C01807=1145.938,166.654,-59.645,-178.486,7.082,148.879
C01808=1145.942,166.405,-59.623,-178.489,7.080,148.879
C01809=1145.947,166.156,-59.601,-178.492,7.077,148.880
C01810=1145.951,165.907,-59.579,-178.495,7.076,148.880
C01811=1145.956,165.658,-59.558,-178.497,7.074,148.880
C01812=1145.961,165.409,-59.535,-178.500,7.071,148.881
C01813=1145.966,165.160,-59.513,-178.503,7.069,148.881
C01814=1145.970,164.911,-59.491,-178.506,7.068,148.881
C01815=1145.975,164.662,-59.469,-178.509,7.065,148.882
C01816=1145.980,164.413,-59.447,-178.511,7.063,148.882
C01817=1145.984,164.165,-59.425,-178.514,7.061,148.882
C01818=1145.988,163.915,-59.403,-178.517,7.059,148.883
C01819=1145.993,163.667,-59.381,-178.520,7.057,148.883
C01820=1145.998,163.417,-59.359,-178.522,7.055,148.883
C01821=1146.003,163.168,-59.337,-178.525,7.052,148.883
C01822=1146.008,162.919,-59.316,-178.528,7.051,148.884
C01823=1146.013,162.670,-59.294,-178.531,7.049,148.884
C01824=1146.017,162.421,-59.272,-178.534,7.046,148.885
C01825=1146.022,162.172,-59.250,-178.536,7.044,148.885
C01826=1146.027,161.923,-59.229,-178.539,7.043,148.885
C01827=1146.031,161.674,-59.206,-178.542,7.040,148.885
C01828=1146.036,161.425,-59.185,-178.545,7.038,148.886
C01829=1146.040,161.176,-59.163,-178.548,7.037,148.886
C01830=1146.045,160.927,-59.141,-178.550,7.034,148.886
C01831=1146.050,160.679,-59.119,-178.553,7.032,148.887
C01832=1146.054,160.429,-59.097,-178.556,7.030,148.887
C01833=1146.059,160.180,-59.076,-178.559,7.029,148.887
C01834=1146.064,159.931,-59.054,-178.562,7.026,148.888
C01835=1146.068,159.682,-59.033,-178.564,7.024,148.888
C01836=1146.073,159.433,-59.011,-178.567,7.022,148.888
C01837=1146.078,159.184,-58.989,-178.570,7.020,148.889
C01838=1146.083,158.935,-58.968,-178.573,7.018,148.889
C01839=1146.088,158.686,-58.946,-178.575,7.016,148.889
C01840=1146.092,158.437,-58.924,-178.578,7.013,148.890
C01841=1146.097,158.188,-58.903,-178.581,7.012,148.890
C01842=1146.101,157.919,-58.880,-178.584,7.010,148.890
C01843=1146.107,157.650,-58.856,-178.587,7.007,148.891
C01844=1146.111,157.381,-58.833,-178.590,7.006,148.891
C01845=1146.117,157.112,-58.810,-178.593,7.003,148.891
C01846=1146.122,156.863,-58.788,-178.596,7.001,148.892
C01847=1146.126,156.613,-58.767,-178.599,6.999,148.892
C01848=1146.130,156.365,-58.745,-178.602,6.997,148.893
C01849=1146.135,156.116,-58.724,-178.604,6.995,148.893
C01850=1146.140,155.867,-58.703,-178.607,6.993,148.893
C01851=1146.145,155.618,-58.681,-178.610,6.991,148.893
C01852=1146.150,155.369,-58.660,-178.613,6.989,148.894
C01853=1146.155,155.120,-58.638,-178.615,6.987,148.894
C01854=1146.159,154.871,-58.616,-178.618,6.986,148.895
C01855=1146.163,154.622,-58.596,-178.621,6.983,148.895
C01856=1146.168,154.373,-58.574,-178.624,6.981,148.895
C01857=1146.174,154.124,-58.553,-178.626,6.979,148.895
C01858=1146.178,153.874,-58.531,-178.629,6.978,148.896
C01859=1146.183,153.625,-58.510,-178.632,6.975,148.896
C01860=1146.187,153.377,-58.489,-178.635,6.973,148.897
C01861=1146.192,153.128,-58.468,-178.638,6.972,148.897
C01862=1146.197,152.878,-58.446,-178.640,6.970,148.897
C01863=1146.202,152.629,-58.425,-178.643,6.967,148.898
C01864=1146.207,152.380,-58.403,-178.646,6.965,148.898
C01865=1146.211,152.131,-58.383,-178.649,6.964,148.898
C01866=1146.215,151.882,-58.361,-178.651,6.962,148.899
C01867=1146.220,151.633,-58.340,-178.655,6.959,148.899
C01868=1146.225,151.384,-58.319,-178.657,6.958,148.899
C01869=1146.230,151.135,-58.298,-178.660,6.956,148.900
C01870=1146.235,150.886,-58.277,-178.662,6.954,148.900
C01871=1146.239,150.637,-58.255,-178.666,6.951,148.900
C01872=1146.244,150.388,-58.234,-178.668,6.950,148.901
C01873=1146.249,150.138,-58.213,-178.671,6.948,148.901
C01874=1146.254,149.890,-58.192,-178.674,6.946,148.901
C01875=1146.258,149.641,-58.171,-178.676,6.945,148.902
C01876=1146.263,149.392,-58.150,-178.680,6.942,148.902
C01877=1146.268,149.142,-58.128,-178.682,6.940,148.902
C01878=1146.272,148.893,-58.108,-178.685,6.938,148.903
C01879=1146.277,148.644,-58.087,-178.687,6.936,148.903
C01880=1146.282,148.395,-58.065,-178.690,6.935,148.904
C01881=1146.286,148.146,-58.045,-178.693,6.932,148.904
C01882=1146.292,147.897,-58.024,-178.696,6.931,148.904
C01883=1146.296,147.648,-58.004,-178.699,6.929,148.905
C01884=1146.300,147.399,-57.982,-178.701,6.927,148.905
C01885=1146.306,147.150,-57.961,-178.705,6.925,148.905
C01886=1146.310,146.901,-57.940,-178.707,6.923,148.906
C01887=1146.315,146.651,-57.919,-178.710,6.921,148.906
C01888=1146.319,146.403,-57.898,-178.712,6.919,148.906
C01889=1146.324,146.154,-57.877,-178.715,6.917,148.907
C01890=1146.329,145.905,-57.857,-178.718,6.916,148.907
C01891=1146.334,145.656,-57.836,-178.721,6.913,148.907
C01892=1146.339,145.407,-57.816,-178.724,6.911,148.908
C01893=1146.344,145.157,-57.795,-178.727,6.910,148.908
C01894=1146.348,144.907,-57.773,-178.729,6.908,148.909
C01895=1146.352,144.659,-57.752,-178.732,6.906,148.909
C01896=1146.358,144.410,-57.731,-178.735,6.904,148.909
C01897=1146.362,144.161,-57.711,-178.738,6.902,148.910
C01898=1146.366,143.912,-57.690,-178.740,6.900,148.910
C01899=1146.372,143.663,-57.670,-178.743,6.898,148.910
C01900=1146.376,143.414,-57.649,-178.746,6.897,148.911
C01901=1146.381,143.164,-57.628,-178.748,6.895,148.911
C01902=1146.386,142.916,-57.608,-178.752,6.892,148.912
C01903=1146.391,142.666,-57.587,-178.754,6.891,148.912
C01904=1146.395,142.417,-57.566,-178.757,6.889,148.912
C01905=1146.400,142.168,-57.545,-178.760,6.887,148.913
C01906=1146.405,141.919,-57.525,-178.763,6.885,148.913
C01907=1146.409,141.670,-57.505,-178.765,6.884,148.913
C01908=1146.415,141.421,-57.484,-178.769,6.881,148.914
C01909=1146.419,141.172,-57.463,-178.771,6.879,148.914
C01910=1146.424,140.923,-57.442,-178.774,6.878,148.915
C01911=1146.429,140.674,-57.422,-178.777,6.876,148.915
C01912=1146.433,140.425,-57.402,-178.779,6.874,148.915
C01913=1146.438,140.176,-57.381,-178.782,6.873,148.916
C01914=1146.443,139.926,-57.361,-178.784,6.871,148.916
C01915=1146.447,139.677,-57.341,-178.788,6.868,148.916
C01916=1146.453,139.428,-57.320,-178.790,6.866,148.917
C01917=1146.457,139.179,-57.299,-178.793,6.865,148.917
C01918=1146.461,138.930,-57.279,-178.796,6.863,148.917
C01919=1146.467,138.681,-57.258,-178.799,6.861,148.918
C01920=1146.471,138.432,-57.238,-178.801,6.859,148.918
C01921=1146.476,138.182,-57.218,-178.804,6.858,148.919
C01922=1146.481,137.933,-57.197,-178.807,6.855,148.919
C01923=1146.485,137.684,-57.177,-178.810,6.854,148.919
C01924=1146.490,137.435,-57.156,-178.813,6.852,148.920
C01925=1146.494,137.186,-57.136,-178.815,6.850,148.920
C01926=1146.500,136.936,-57.116,-178.818,6.848,148.921
C01927=1146.505,136.688,-57.096,-178.821,6.847,148.921
C01928=1146.509,136.439,-57.075,-178.824,6.845,148.921
C01929=1146.515,136.189,-57.055,-178.826,6.843,148.922
C01930=1146.519,135.940,-57.035,-178.830,6.841,148.922
C01931=1146.524,135.691,-57.014,-178.832,6.839,148.923
C01932=1146.528,135.442,-56.994,-178.835,6.837,148.923
C01933=1146.533,135.193,-56.974,-178.838,6.836,148.923
C01934=1146.538,134.943,-56.953,-178.840,6.834,148.924
C01935=1146.542,134.694,-56.933,-178.843,6.832,148.924
C01936=1146.548,134.446,-56.914,-178.846,6.831,148.925
C01937=1146.552,134.197,-56.893,-178.849,6.829,148.925
C01938=1146.557,133.947,-56.874,-178.851,6.827,148.925
C01939=1146.562,133.698,-56.853,-178.854,6.825,148.926
C01940=1146.566,133.449,-56.832,-178.857,6.823,148.926
C01941=1146.571,133.199,-56.813,-178.860,6.821,148.926
C01942=1146.576,132.950,-56.792,-178.863,6.819,148.927
C01943=1146.581,132.701,-56.773,-178.865,6.818,148.927
C01944=1146.585,132.452,-56.753,-178.868,6.816,148.928
C01945=1146.590,132.203,-56.733,-178.871,6.814,148.928
C01946=1146.596,131.935,-56.711,-178.874,6.813,148.928
C01947=1146.600,131.666,-56.689,-178.877,6.810,148.929
C01948=1146.606,131.397,-56.668,-178.880,6.808,148.929
C01949=1146.611,131.129,-56.646,-178.882,6.807,148.930
C01950=1146.615,130.879,-56.626,-178.885,6.805,148.930
C01951=1146.620,130.630,-56.606,-178.888,6.803,148.930
C01952=1146.625,130.382,-56.587,-178.890,6.802,148.931
C01953=1146.630,130.133,-56.566,-178.894,6.799,148.931
C01954=1146.635,129.883,-56.546,-178.897,6.797,148.932
C01955=1146.640,129.633,-56.526,-178.900,6.796,148.932
C01956=1146.645,129.385,-56.506,-178.902,6.794,148.933
C01957=1146.650,129.135,-56.487,-178.905,6.793,148.933
C01958=1146.654,128.886,-56.466,-178.908,6.791,148.933
C01959=1146.659,128.637,-56.447,-178.911,6.789,148.934
C01960=1146.664,128.388,-56.427,-178.913,6.788,148.934
C01961=1146.669,128.139,-56.407,-178.916,6.786,148.935
C01962=1146.673,127.889,-56.387,-178.919,6.784,148.935
C01963=1146.678,127.640,-56.368,-178.921,6.782,148.935
C01964=1146.683,127.392,-56.348,-178.924,6.781,148.936
C01965=1146.688,127.142,-56.328,-178.927,6.779,148.936
C01966=1146.693,126.892,-56.308,-178.930,6.777,148.937
C01967=1146.696,126.644,-56.289,-178.932,6.776,148.937
C01968=1146.702,126.395,-56.269,-178.935,6.774,148.937
C01969=1146.706,126.145,-56.250,-178.938,6.772,148.938
C01970=1146.711,125.896,-56.230,-178.940,6.771,148.938
C01971=1146.716,125.648,-56.210,-178.943,6.769,148.939
C01972=1146.721,125.398,-56.190,-178.947,6.766,148.939
C01973=1146.726,125.148,-56.171,-178.949,6.765,148.939
C01974=1146.731,124.900,-56.151,-178.952,6.763,148.940
C01975=1146.735,124.651,-56.131,-178.955,6.761,148.940
C01976=1146.740,124.401,-56.111,-178.957,6.760,148.941
C01977=1146.746,124.152,-56.092,-178.960,6.758,148.941
C01978=1146.750,123.903,-56.073,-178.963,6.756,148.941
C01979=1146.754,123.653,-56.053,-178.966,6.754,148.942
C01980=1146.760,123.404,-56.034,-178.969,6.753,148.942
C01981=1146.764,123.156,-56.014,-178.971,6.751,148.943
C01982=1146.769,122.906,-55.994,-178.974,6.750,148.943
C01983=1146.774,122.657,-55.975,-178.977,6.748,148.944
C01984=1146.778,122.408,-55.956,-178.980,6.746,148.944
C01985=1146.783,122.158,-55.936,-178.982,6.745,148.944
C01986=1146.788,121.909,-55.917,-178.985,6.743,148.945
C01987=1146.793,121.660,-55.897,-178.988,6.741,148.945
C01988=1146.798,121.411,-55.878,-178.991,6.739,148.946
C01989=1146.802,121.162,-55.859,-178.993,6.738,148.946
C01990=1146.807,120.912,-55.839,-178.996,6.736,148.946
C01991=1146.812,120.663,-55.820,-178.999,6.734,148.947
C01992=1146.817,120.414,-55.800,-179.001,6.733,148.947
C01993=1146.822,120.165,-55.781,-179.004,6.731,148.948
C01994=1146.827,119.916,-55.762,-179.007,6.730,148.948
C01995=1146.831,119.666,-55.742,-179.010,6.728,148.949
C01996=1146.837,119.417,-55.723,-179.013,6.726,148.949
C01997=1146.841,119.168,-55.704,-179.016,6.725,148.949
C01998=1146.846,118.919,-55.684,-179.018,6.723,148.950
C01999=1146.851,118.669,-55.665,-179.021,6.721,148.950
C02000=1146.856,118.421,-55.646,-179.024,6.719,148.951
C02001=1146.860,118.171,-55.626,-179.026,6.718,148.951
C02002=1146.865,117.922,-55.607,-179.029,6.716,148.951
C02003=1146.870,117.673,-55.588,-179.032,6.714,148.952
C02004=1146.874,117.423,-55.569,-179.035,6.713,148.952
C02005=1146.880,117.174,-55.550,-179.038,6.711,148.953
C02006=1146.885,116.925,-55.530,-179.040,6.710,148.953
C02007=1146.889,116.676,-55.512,-179.043,6.709,148.954
C02008=1146.894,116.426,-55.492,-179.045,6.707,148.954
C02009=1146.899,116.178,-55.473,-179.048,6.705,148.954
C02010=1146.903,115.928,-55.454,-179.051,6.704,148.955
C02011=1146.909,115.679,-55.435,-179.054,6.702,148.955
C02012=1146.913,115.430,-55.416,-179.056,6.700,148.956
C02013=1146.918,115.181,-55.397,-179.059,6.699,148.956
C02014=1146.923,114.931,-55.377,-179.062,6.697,148.956
C02015=1146.928,114.682,-55.359,-179.065,6.696,148.957
C02016=1146.933,114.432,-55.339,-179.068,6.694,148.958
C02017=1146.937,114.184,-55.321,-179.070,6.692,148.958
C02018=1146.943,113.935,-55.301,-179.073,6.690,148.958
C02019=1146.948,113.685,-55.282,-179.076,6.689,148.959
C02020=1146.952,113.436,-55.264,-179.079,6.687,148.959
C02021=1146.957,113.187,-55.244,-179.081,6.685,148.960
C02022=1146.962,112.937,-55.226,-179.084,6.684,148.960
C02023=1146.967,112.688,-55.206,-179.087,6.682,148.960
C02024=1146.971,112.439,-55.188,-179.090,6.681,148.961
C02025=1146.976,112.189,-55.169,-179.093,6.679,148.961
C02026=1146.981,111.941,-55.150,-179.095,6.678,148.962
C02027=1146.986,111.692,-55.131,-179.098,6.676,148.962
C02028=1146.991,111.442,-55.112,-179.100,6.675,148.963
C02029=1146.996,111.193,-55.093,-179.103,6.673,148.963
C02030=1147.000,110.943,-55.075,-179.106,6.671,148.963
C02031=1147.006,110.694,-55.055,-179.109,6.670,148.964
C02032=1147.010,110.446,-55.037,-179.112,6.668,148.964
C02033=1147.015,110.196,-55.018,-179.114,6.667,148.965
C02034=1147.020,109.947,-54.999,-179.117,6.665,148.965
C02035=1147.025,109.697,-54.980,-179.120,6.663,148.966
C02036=1147.029,109.448,-54.962,-179.123,6.662,148.966
C02037=1147.034,109.199,-54.944,-179.125,6.660,148.967
C02038=1147.039,108.949,-54.924,-179.128,6.659,148.967
C02039=1147.044,108.700,-54.906,-179.131,6.658,148.968
C02040=1147.049,108.451,-54.887,-179.133,6.656,148.968
C02041=1147.054,108.202,-54.868,-179.136,6.654,148.968
C02042=1147.058,107.953,-54.850,-179.139,6.653,148.969
C02043=1147.063,107.703,-54.831,-179.142,6.651,148.969
C02044=1147.068,107.454,-54.812,-179.144,6.649,148.970
C02045=1147.074,107.205,-54.793,-179.147,6.648,148.970
C02046=1147.078,106.955,-54.775,-179.150,6.646,148.971
C02047=1147.083,106.706,-54.756,-179.153,6.644,148.971
C02048=1147.088,106.457,-54.738,-179.155,6.644,148.971
C02049=1147.092,106.208,-54.719,-179.158,6.642,148.972
C02050=1147.097,105.939,-54.699,-179.161,6.641,148.973
C02051=1147.103,105.671,-54.679,-179.164,6.638,148.973
C02052=1147.108,105.403,-54.660,-179.167,6.636,148.973
C02053=1147.114,105.135,-54.639,-179.170,6.635,148.974
C02054=1147.118,104.885,-54.621,-179.173,6.633,148.974
C02055=1147.123,104.636,-54.603,-179.176,6.632,148.975
C02056=1147.128,104.387,-54.584,-179.178,6.631,148.975
C02057=1147.133,104.137,-54.566,-179.181,6.629,148.976
C02058=1147.137,103.888,-54.547,-179.183,6.627,148.976
C02059=1147.142,103.639,-54.529,-179.186,6.626,148.977
C02060=1147.148,103.390,-54.510,-179.189,6.624,148.977
C02061=1147.152,103.140,-54.492,-179.192,6.623,148.978
C02062=1147.157,102.891,-54.474,-179.195,6.621,148.978
C02063=1147.162,102.642,-54.455,-179.197,6.620,148.978
C02064=1147.167,102.392,-54.436,-179.200,6.619,148.979
C02065=1147.172,102.143,-54.418,-179.203,6.617,148.979
C02066=1147.176,101.893,-54.400,-179.205,6.616,148.980
C02067=1147.181,101.644,-54.382,-179.208,6.614,148.980
C02068=1147.187,101.395,-54.363,-179.211,6.612,148.981
C02069=1147.192,101.146,-54.345,-179.214,6.610,148.981
C02070=1147.196,100.896,-54.326,-179.216,6.610,148.981
C02071=1147.201,100.647,-54.308,-179.219,6.608,148.982
C02072=1147.206,100.398,-54.290,-179.222,6.607,148.983
C02073=1147.211,100.149,-54.272,-179.224,6.605,148.983
C02074=1147.216,99.899,-54.254,-179.227,6.603,148.983
C02075=1147.220,99.650,-54.235,-179.230,6.602,148.984
C02076=1147.225,99.401,-54.217,-179.233,6.600,148.984
C02077=1147.230,99.152,-54.199,-179.235,6.599,148.985
C02078=1147.235,98.903,-54.181,-179.238,6.598,148.985
C02079=1147.240,98.653,-54.163,-179.241,6.596,148.986
C02080=1147.244,98.403,-54.145,-179.244,6.594,148.986
C02081=1147.249,98.154,-54.127,-179.247,6.593,148.987
C02082=1147.254,97.905,-54.109,-179.249,6.592,148.987
C02083=1147.260,97.656,-54.090,-179.252,6.590,148.988
C02084=1147.265,97.406,-54.072,-179.254,6.589,148.988
C02085=1147.270,97.157,-54.054,-179.257,6.587,148.988
C02086=1147.274,96.908,-54.036,-179.260,6.586,148.989
C02087=1147.279,96.658,-54.018,-179.263,6.584,148.989
C02088=1147.284,96.409,-54.000,-179.265,6.583,148.990
C02089=1147.289,96.160,-53.982,-179.268,6.581,148.990
C02090=1147.294,95.911,-53.964,-179.271,6.580,148.991
C02091=1147.298,95.662,-53.946,-179.274,6.578,148.991
C02092=1147.303,95.412,-53.928,-179.277,6.577,148.992
C02093=1147.308,95.163,-53.910,-179.279,6.576,148.992
C02094=1147.313,94.914,-53.892,-179.281,6.574,148.993
C02095=1147.317,94.664,-53.874,-179.285,6.573,148.993
C02096=1147.323,94.414,-53.856,-179.287,6.571,148.994
C02097=1147.328,94.165,-53.838,-179.290,6.570,148.994
C02098=1147.333,93.916,-53.820,-179.292,6.569,148.994
C02099=1147.337,93.667,-53.802,-179.295,6.567,148.995
C02100=1147.342,93.418,-53.784,-179.298,6.566,148.996
C02101=1147.347,93.168,-53.766,-179.301,6.564,148.996
C02102=1147.352,92.919,-53.749,-179.304,6.562,148.996
C02103=1147.357,92.669,-53.731,-179.306,6.561,148.997
C02104=1147.362,92.420,-53.713,-179.309,6.560,148.997
C02105=1147.367,92.171,-53.695,-179.312,6.558,148.998
C02106=1147.372,91.922,-53.677,-179.314,6.557,148.998
C02107=1147.377,91.672,-53.660,-179.317,6.555,148.999
C02108=1147.382,91.423,-53.643,-179.319,6.554,148.999
C02109=1147.386,91.174,-53.625,-179.323,6.553,149.000
C02110=1147.391,90.925,-53.607,-179.325,6.551,149.000
C02111=1147.397,90.675,-53.589,-179.328,6.550,149.001
C02112=1147.401,90.426,-53.571,-179.330,6.549,149.001
C02113=1147.406,90.177,-53.553,-179.333,6.547,149.002
C02114=1147.411,89.928,-53.535,-179.336,6.546,149.002
C02115=1147.417,89.678,-53.518,-179.339,6.544,149.003
C02116=1147.421,89.429,-53.501,-179.341,6.543,149.003
C02117=1147.426,89.180,-53.483,-179.344,6.542,149.004
C02118=1147.431,88.930,-53.465,-179.347,6.540,149.004
C02119=1147.436,88.681,-53.448,-179.350,6.538,149.004
C02120=1147.441,88.432,-53.430,-179.352,6.537,149.005
C02121=1147.446,88.182,-53.412,-179.355,6.536,149.006
C02122=1147.450,87.933,-53.395,-179.358,6.535,149.006
C02123=1147.455,87.683,-53.378,-179.361,6.533,149.006
C02124=1147.460,87.434,-53.360,-179.363,6.531,149.007
C02125=1147.465,87.185,-53.342,-179.366,6.531,149.007
C02126=1147.470,86.935,-53.325,-179.369,6.529,149.008
C02127=1147.474,86.686,-53.307,-179.371,6.527,149.008
C02128=1147.480,86.436,-53.290,-179.374,6.526,149.009
C02129=1147.485,86.187,-53.272,-179.377,6.525,149.009
C02130=1147.490,85.937,-53.255,-179.379,6.524,149.010
C02131=1147.494,85.689,-53.237,-179.382,6.522,149.010
C02132=1147.499,85.439,-53.220,-179.384,6.521,149.011
C02133=1147.504,85.190,-53.202,-179.388,6.520,149.011
C02134=1147.509,84.940,-53.185,-179.390,6.518,149.012
C02135=1147.514,84.691,-53.167,-179.393,6.516,149.012
C02136=1147.519,84.442,-53.150,-179.395,6.516,149.013
C02137=1147.524,84.193,-53.132,-179.398,6.514,149.013
C02138=1147.529,83.943,-53.116,-179.401,6.513,149.014
C02139=1147.534,83.694,-53.098,-179.404,6.511,149.014
C02140=1147.539,83.444,-53.080,-179.407,6.510,149.015
C02141=1147.543,83.195,-53.063,-179.409,6.509,149.015
C02142=1147.548,82.946,-53.046,-179.412,6.507,149.016
C02143=1147.553,82.696,-53.029,-179.414,6.506,149.016
C02144=1147.558,82.447,-53.011,-179.417,6.505,149.017
C02145=1147.563,82.198,-52.994,-179.420,6.503,149.017
C02146=1147.569,81.948,-52.977,-179.423,6.502,149.017
C02147=1147.573,81.699,-52.960,-179.425,6.501,149.018
C02148=1147.578,81.449,-52.942,-179.428,6.499,149.019
C02149=1147.583,81.200,-52.926,-179.431,6.498,149.019
C02150=1147.587,80.951,-52.908,-179.433,6.497,149.019
C02151=1147.593,80.702,-52.891,-179.436,6.495,149.020
C02152=1147.598,80.452,-52.874,-179.439,6.494,149.020
C02153=1147.603,80.203,-52.856,-179.441,6.493,149.021
C02154=1147.607,79.934,-52.838,-179.444,6.492,149.022
C02155=1147.613,79.666,-52.820,-179.447,6.490,149.022
C02156=1147.619,79.397,-52.801,-179.450,6.489,149.023
C02157=1147.623,79.129,-52.783,-179.453,6.487,149.023
C02158=1147.629,78.880,-52.765,-179.456,6.485,149.023
C02159=1147.633,78.631,-52.749,-179.459,6.485,149.024
C02160=1147.639,78.381,-52.731,-179.461,6.483,149.025
C02161=1147.644,78.131,-52.714,-179.464,6.482,149.025
C02162=1147.648,77.882,-52.697,-179.466,6.481,149.025
C02163=1147.654,77.633,-52.680,-179.469,6.479,149.026
C02164=1147.658,77.384,-52.663,-179.472,6.478,149.027
C02165=1147.663,77.134,-52.646,-179.474,6.477,149.027
C02166=1147.668,76.884,-52.629,-179.477,6.476,149.028
C02167=1147.674,76.635,-52.612,-179.480,6.474,149.028
C02168=1147.678,76.386,-52.596,-179.483,6.472,149.028
C02169=1147.683,76.137,-52.578,-179.485,6.471,149.029
C02170=1147.688,75.887,-52.561,-179.488,6.470,149.030
C02171=1147.693,75.638,-52.545,-179.491,6.468,149.030
C02172=1147.698,75.389,-52.527,-179.493,6.467,149.030
C02173=1147.702,75.139,-52.511,-179.496,6.466,149.031
C02174=1147.708,74.889,-52.493,-179.499,6.465,149.031
C02175=1147.713,74.641,-52.477,-179.501,6.464,149.032
C02176=1147.718,74.391,-52.460,-179.505,6.462,149.033
C02177=1147.722,74.141,-52.443,-179.507,6.461,149.033
C02178=1147.727,73.892,-52.427,-179.509,6.460,149.033
C02179=1147.733,73.643,-52.410,-179.513,6.459,149.034
C02180=1147.737,73.393,-52.393,-179.515,6.458,149.035
C02181=1147.742,73.143,-52.376,-179.518,6.456,149.035
C02182=1147.747,72.895,-52.359,-179.520,6.454,149.035
C02183=1147.752,72.645,-52.343,-179.523,6.454,149.036
C02184=1147.757,72.395,-52.326,-179.526,6.452,149.036
C02185=1147.762,72.147,-52.309,-179.528,6.451,149.037
C02186=1147.767,71.897,-52.293,-179.531,6.450,149.038
C02187=1147.772,71.647,-52.275,-179.534,6.448,149.038
C02188=1147.777,71.399,-52.259,-179.537,6.447,149.038
C02189=1147.782,71.149,-52.242,-179.539,6.446,149.039
C02190=1147.787,70.899,-52.225,-179.542,6.445,149.040
C02191=1147.792,70.650,-52.209,-179.544,6.444,149.040
C02192=1147.796,70.401,-52.192,-179.547,6.442,149.041
C02193=1147.802,70.151,-52.175,-179.550,6.441,149.041
C02194=1147.807,69.902,-52.159,-179.552,6.440,149.041
C02195=1147.811,69.652,-52.143,-179.555,6.439,149.042
C02196=1147.817,69.403,-52.125,-179.558,6.437,149.043
C02197=1147.822,69.154,-52.109,-179.560,6.436,149.043
C02198=1147.826,68.904,-52.092,-179.564,6.435,149.044
C02199=1147.831,68.655,-52.076,-179.566,6.434,149.044
C02200=1147.836,68.406,-52.059,-179.568,6.432,149.045
C02201=1147.841,68.156,-52.043,-179.572,6.431,149.045
C02202=1147.846,67.907,-52.026,-179.574,6.430,149.046
C02203=1147.851,67.657,-52.010,-179.577,6.428,149.046
C02204=1147.857,67.408,-51.993,-179.579,6.428,149.047
C02205=1147.861,67.159,-51.976,-179.582,6.426,149.047
C02206=1147.866,66.909,-51.960,-179.585,6.425,149.048
C02207=1147.871,66.660,-51.944,-179.587,6.424,149.048
C02208=1147.875,66.410,-51.927,-179.590,6.422,149.049
C02209=1147.881,66.161,-51.910,-179.592,6.422,149.049
C02210=1147.886,65.911,-51.894,-179.595,6.420,149.050
C02211=1147.891,65.662,-51.878,-179.598,6.419,149.050
C02212=1147.896,65.413,-51.861,-179.600,6.418,149.051
C02213=1147.900,65.163,-51.846,-179.604,6.417,149.051
C02214=1147.905,64.914,-51.829,-179.606,6.416,149.052
C02215=1147.911,64.664,-51.812,-179.608,6.414,149.052
C02216=1147.916,64.415,-51.796,-179.612,6.413,149.053
C02217=1147.921,64.165,-51.780,-179.614,6.412,149.053
C02218=1147.926,63.917,-51.763,-179.617,6.410,149.054
C02219=1147.930,63.666,-51.747,-179.619,6.410,149.054
C02220=1147.936,63.418,-51.731,-179.622,6.408,149.055
C02221=1147.940,63.168,-51.714,-179.624,6.407,149.055
C02222=1147.945,62.919,-51.699,-179.627,6.406,149.056
C02223=1147.951,62.669,-51.682,-179.630,6.404,149.056
C02224=1147.956,62.420,-51.666,-179.632,6.403,149.057
C02225=1147.960,62.170,-51.649,-179.635,6.402,149.057
C02226=1147.966,61.921,-51.634,-179.638,6.401,149.058
C02227=1147.970,61.671,-51.617,-179.640,6.400,149.058
C02228=1147.975,61.422,-51.601,-179.643,6.399,149.059
C02229=1147.980,61.172,-51.585,-179.646,6.397,149.059
C02230=1147.985,60.924,-51.569,-179.648,6.397,149.060
C02231=1147.990,60.673,-51.553,-179.651,6.395,149.061
C02232=1147.995,60.425,-51.536,-179.654,6.394,149.061
C02233=1148.000,60.175,-51.520,-179.657,6.393,149.062
C02234=1148.005,59.926,-51.504,-179.659,6.392,149.062
C02235=1148.010,59.676,-51.488,-179.661,6.391,149.062
C02236=1148.015,59.427,-51.472,-179.665,6.389,149.063
C02237=1148.020,59.177,-51.456,-179.667,6.389,149.064
C02238=1148.025,58.927,-51.440,-179.670,6.387,149.064
C02239=1148.030,58.679,-51.424,-179.672,6.386,149.065
C02240=1148.035,58.428,-51.408,-179.675,6.385,149.065
C02241=1148.040,58.180,-51.392,-179.678,6.383,149.066
C02242=1148.045,57.930,-51.376,-179.680,6.383,149.066
C02243=1148.050,57.681,-51.359,-179.683,6.381,149.067
C02244=1148.055,57.431,-51.344,-179.685,6.380,149.067
C02245=1148.060,57.181,-51.328,-179.688,6.379,149.068
C02246=1148.065,56.933,-51.312,-179.691,6.378,149.068
C02247=1148.070,56.682,-51.296,-179.694,6.377,149.069
C02248=1148.075,56.433,-51.280,-179.696,6.376,149.069
C02249=1148.080,56.184,-51.264,-179.699,6.374,149.070
C02250=1148.085,55.934,-51.248,-179.701,6.374,149.070
C02251=1148.091,55.685,-51.232,-179.704,6.372,149.071
C02252=1148.095,55.435,-51.216,-179.706,6.371,149.071
C02253=1148.100,55.186,-51.201,-179.710,6.370,149.072
C02254=1148.105,54.937,-51.185,-179.712,6.369,149.072
C02255=1148.110,54.687,-51.168,-179.715,6.368,149.073
C02256=1148.115,54.438,-51.153,-179.717,6.367,149.074
C02257=1148.120,54.188,-51.137,-179.720,6.365,149.074
C02258=1148.125,53.919,-51.120,-179.723,6.364,149.075
C02259=1148.131,53.651,-51.103,-179.725,6.363,149.075
C02260=1148.136,53.382,-51.086,-179.728,6.362,149.076
C02261=1148.142,53.114,-51.069,-179.732,6.361,149.076
C02262=1148.147,52.865,-51.054,-179.734,6.360,149.077
C02263=1148.151,52.615,-51.038,-179.737,6.358,149.077
C02264=1148.157,52.365,-51.022,-179.739,6.358,149.078
C02265=1148.162,52.116,-51.006,-179.742,6.356,149.078
C02266=1148.167,51.866,-50.990,-179.744,6.355,149.079
C02267=1148.172,51.617,-50.974,-179.747,6.354,149.080
C02268=1148.177,51.368,-50.959,-179.750,6.353,149.080
C02269=1148.181,51.118,-50.943,-179.753,6.352,149.081
C02270=1148.187,50.868,-50.928,-179.755,6.351,149.081
C02271=1148.192,50.620,-50.911,-179.758,6.349,149.082
C02272=1148.196,50.370,-50.896,-179.760,6.349,149.082
C02273=1148.201,50.120,-50.881,-179.763,6.347,149.083
C02274=1148.207,49.871,-50.865,-179.765,6.346,149.083
C02275=1148.212,49.622,-50.849,-179.768,6.345,149.084
C02276=1148.216,49.372,-50.834,-179.771,6.344,149.084
C02277=1148.222,49.122,-50.818,-179.774,6.343,149.085
C02278=1148.227,48.873,-50.803,-179.776,6.342,149.085
C02279=1148.232,48.624,-50.787,-179.779,6.340,149.086
C02280=1148.236,48.374,-50.772,-179.781,6.340,149.086
C02281=1148.242,48.124,-50.756,-179.784,6.339,149.087
C02282=1148.247,47.875,-50.741,-179.787,6.338,149.088
C02283=1148.252,47.626,-50.726,-179.789,6.337,149.088
C02284=1148.257,47.376,-50.710,-179.792,6.335,149.088
C02285=1148.262,47.126,-50.694,-179.794,6.335,149.089
C02286=1148.267,46.877,-50.679,-179.797,6.333,149.090
C02287=1148.272,46.628,-50.664,-179.800,6.333,149.090
C02288=1148.277,46.378,-50.648,-179.803,6.331,149.091
C02289=1148.281,46.129,-50.633,-179.805,6.330,149.091
C02290=1148.287,45.879,-50.617,-179.808,6.329,149.092
C02291=1148.292,45.630,-50.601,-179.810,6.328,149.092
C02292=1148.297,45.381,-50.586,-179.813,6.328,149.093
C02293=1148.302,45.131,-50.570,-179.815,6.326,149.093
C02294=1148.306,44.882,-50.556,-179.818,6.325,149.094
C02295=1148.312,44.632,-50.540,-179.821,6.324,149.094
C02296=1148.317,44.383,-50.524,-179.823,6.323,149.095
C02297=1148.322,44.133,-50.510,-179.826,6.322,149.096
C02298=1148.327,43.884,-50.494,-179.828,6.321,149.096
C02299=1148.331,43.634,-50.479,-179.831,6.319,149.096
C02300=1148.337,43.384,-50.464,-179.834,6.319,149.097
C02301=1148.342,43.135,-50.448,-179.836,6.318,149.098
C02302=1148.347,42.886,-50.433,-179.839,6.317,149.098
C02303=1148.353,42.636,-50.418,-179.841,6.316,149.099
C02304=1148.357,42.387,-50.403,-179.844,6.314,149.099
C02305=1148.362,42.137,-50.387,-179.847,6.314,149.100
C02306=1148.367,41.888,-50.372,-179.850,6.312,149.100
C02307=1148.372,41.638,-50.357,-179.852,6.312,149.101
C02308=1148.377,41.389,-50.342,-179.854,6.311,149.101
C02309=1148.382,41.139,-50.327,-179.857,6.309,149.102
C02310=1148.388,40.890,-50.311,-179.860,6.309,149.102
C02311=1148.392,40.641,-50.296,-179.862,6.307,149.103
C02312=1148.398,40.391,-50.281,-179.865,6.307,149.104
C02313=1148.402,40.141,-50.266,-179.868,6.305,149.104
C02314=1148.408,39.891,-50.250,-179.870,6.304,149.104
C02315=1148.412,39.642,-50.235,-179.873,6.304,149.105
C02316=1148.418,39.392,-50.220,-179.875,6.302,149.106
C02317=1148.423,39.143,-50.205,-179.878,6.302,149.106
C02318=1148.427,38.894,-50.190,-179.881,6.300,149.107
C02319=1148.433,38.644,-50.176,-179.883,6.299,149.107
C02320=1148.438,38.395,-50.161,-179.886,6.299,149.108
C02321=1148.443,38.146,-50.145,-179.888,6.297,149.108
C02322=1148.448,37.896,-50.131,-179.891,6.296,149.109
C02323=1148.453,37.647,-50.115,-179.894,6.295,149.109
C02324=1148.458,37.397,-50.101,-179.896,6.294,149.110
C02325=1148.464,37.147,-50.085,-179.899,6.294,149.111
C02326=1148.468,36.898,-50.070,-179.901,6.292,149.111
C02327=1148.473,36.648,-50.056,-179.904,6.291,149.112
C02328=1148.478,36.399,-50.040,-179.907,6.290,149.112
C02329=1148.483,36.149,-50.026,-179.909,6.289,149.113
C02330=1148.488,35.899,-50.010,-179.912,6.288,149.113
C02331=1148.493,35.650,-49.995,-179.914,6.287,149.114
C02332=1148.498,35.401,-49.981,-179.917,6.286,149.114
C02333=1148.503,35.151,-49.965,-179.920,6.285,149.115
C02334=1148.508,34.901,-49.951,-179.922,6.284,149.115
C02335=1148.513,34.652,-49.936,-179.925,6.283,149.116
C02336=1148.519,34.402,-49.921,-179.928,6.282,149.117
C02337=1148.523,34.153,-49.906,-179.930,6.281,149.117
C02338=1148.528,33.904,-49.892,-179.932,6.280,149.118
C02339=1148.534,33.654,-49.876,-179.935,6.279,149.118
C02340=1148.539,33.404,-49.862,-179.938,6.278,149.119
C02341=1148.543,33.155,-49.847,-179.941,6.277,149.119
C02342=1148.549,32.905,-49.832,-179.943,6.276,149.120
C02343=1148.554,32.656,-49.817,-179.946,6.276,149.120
C02344=1148.559,32.407,-49.803,-179.948,6.274,149.121
C02345=1148.564,32.157,-49.788,-179.951,6.273,149.121
C02346=1148.569,31.907,-49.773,-179.953,6.273,149.122
C02347=1148.574,31.658,-49.759,-179.956,6.271,149.122
C02348=1148.579,31.409,-49.744,-179.959,6.271,149.123
C02349=1148.585,31.159,-49.729,-179.961,6.270,149.124
C02350=1148.590,30.910,-49.715,-179.963,6.268,149.124
C02351=1148.594,30.661,-49.700,-179.966,6.268,149.125
C02352=1148.599,30.411,-49.686,-179.968,6.267,149.125
C02353=1148.605,30.161,-49.671,-179.972,6.266,149.126
C02354=1148.610,29.912,-49.656,-179.974,6.265,149.126
C02355=1148.615,29.662,-49.642,-179.976,6.264,149.127
C02356=1148.619,29.413,-49.627,-179.979,6.263,149.127
C02357=1148.625,29.163,-49.612,-179.981,6.262,149.128
C02358=1148.630,28.913,-49.597,-179.985,6.261,149.129
C02359=1148.635,28.663,-49.583,-179.987,6.260,149.129
C02360=1148.640,28.414,-49.568,-179.989,6.259,149.130
C02361=1148.644,28.165,-49.554,-179.992,6.258,149.130
C02362=1148.651,27.896,-49.538,-179.995,6.257,149.131
C02363=1148.656,27.627,-49.522,-179.998,6.256,149.131
C02364=1148.662,27.358,-49.507,180.000,6.255,149.132
C02365=1148.667,27.089,-49.492,179.997,6.254,149.133
C02366=1148.672,26.839,-49.477,179.994,6.253,149.133
C02367=1148.677,26.590,-49.462,179.992,6.253,149.134
C02368=1148.682,26.340,-49.447,179.989,6.251,149.134
C02369=1148.687,26.091,-49.433,179.987,6.250,149.135
C02370=1148.692,25.842,-49.419,179.984,6.250,149.135
C02371=1148.697,25.592,-49.405,179.982,6.249,149.136
C02372=1148.702,25.342,-49.391,179.979,6.248,149.137
C02373=1148.707,25.093,-49.376,179.977,6.247,149.137
C02374=1148.713,24.843,-49.361,179.974,6.246,149.138
C02375=1148.718,24.593,-49.346,179.971,6.245,149.138
C02376=1148.723,24.344,-49.332,179.969,6.244,149.139
C02377=1148.728,24.095,-49.318,179.966,6.244,149.139
C02378=1148.733,23.845,-49.304,179.964,6.242,149.140
C02379=1148.738,23.595,-49.290,179.961,6.241,149.140
C02380=1148.743,23.346,-49.275,179.959,6.241,149.141
C02381=1148.748,23.097,-49.260,179.956,6.239,149.142
C02382=1148.753,22.848,-49.247,179.953,6.239,149.142
C02383=1148.758,22.598,-49.232,179.951,6.238,149.143
C02384=1148.763,22.348,-49.218,179.949,6.237,149.143
C02385=1148.768,22.098,-49.204,179.946,6.236,149.144
C02386=1148.773,21.849,-49.189,179.943,6.235,149.144
C02387=1148.779,21.600,-49.176,179.941,6.234,149.145
C02388=1148.784,21.350,-49.161,179.938,6.233,149.145
C02389=1148.789,21.100,-49.147,179.936,6.232,149.146
C02390=1148.793,20.851,-49.133,179.933,6.232,149.147
C02391=1148.798,20.601,-49.118,179.930,6.230,149.147
C02392=1148.804,20.352,-49.105,179.928,6.230,149.148
C02393=1148.809,20.102,-49.090,179.925,6.229,149.148
C02394=1148.814,19.852,-49.076,179.923,6.228,149.149
C02395=1148.819,19.603,-49.062,179.920,6.227,149.149
C02396=1148.824,19.354,-49.048,179.918,6.226,149.150
C02397=1148.829,19.104,-49.034,179.915,6.226,149.150
C02398=1148.834,18.854,-49.019,179.913,6.225,149.151
C02399=1148.839,18.605,-49.005,179.910,6.224,149.152
C02400=1148.845,18.356,-48.991,179.908,6.223,149.152
C02401=1148.850,18.106,-48.977,179.905,6.222,149.153
C02402=1148.855,17.856,-48.962,179.902,6.221,149.153
C02403=1148.860,17.607,-48.949,179.900,6.220,149.154
C02404=1148.866,17.357,-48.935,179.897,6.219,149.154
C02405=1148.871,17.107,-48.921,179.895,6.219,149.155
C02406=1148.875,16.858,-48.907,179.892,6.217,149.155
C02407=1148.880,16.609,-48.893,179.890,6.216,149.156
C02408=1148.885,16.359,-48.879,179.887,6.216,149.157
C02409=1148.890,16.109,-48.865,179.885,6.215,149.157
C02410=1148.896,15.860,-48.851,179.882,6.214,149.158
C02411=1148.901,15.610,-48.837,179.879,6.213,149.158
C02412=1148.906,15.360,-48.823,179.877,6.212,149.159
C02413=1148.911,15.110,-48.809,179.875,6.212,149.159
C02414=1148.916,14.862,-48.795,179.872,6.210,149.160
C02415=1148.921,14.612,-48.781,179.869,6.210,149.160
C02416=1148.926,14.362,-48.767,179.867,6.209,149.161
C02417=1148.932,14.113,-48.753,179.864,6.208,149.162
C02418=1148.936,13.863,-48.739,179.862,6.207,149.162
C02419=1148.941,13.613,-48.725,179.859,6.206,149.163
C02420=1148.947,13.364,-48.712,179.857,6.206,149.163
C02421=1148.951,13.114,-48.698,179.854,6.205,149.164
C02422=1148.957,12.865,-48.684,179.851,6.204,149.164
C02423=1148.962,12.616,-48.670,179.849,6.203,149.165
C02424=1148.967,12.365,-48.656,179.847,6.202,149.165
C02425=1148.972,12.117,-48.643,179.844,6.201,149.166
C02426=1148.977,11.867,-48.629,179.842,6.201,149.167
C02427=1148.982,11.616,-48.615,179.839,6.199,149.167
C02428=1148.988,11.367,-48.601,179.836,6.199,149.168
C02429=1148.992,11.118,-48.588,179.834,6.198,149.168
C02430=1148.998,10.869,-48.574,179.832,6.198,149.169
C02431=1149.003,10.619,-48.560,179.829,6.196,149.169
C02432=1149.008,10.369,-48.546,179.827,6.195,149.170
C02433=1149.013,10.120,-48.533,179.824,6.195,149.170
C02434=1149.018,9.870,-48.519,179.822,6.194,149.171
C02435=1149.023,9.621,-48.505,179.819,6.194,149.172
C02436=1149.029,9.371,-48.491,179.816,6.192,149.172
C02437=1149.033,9.121,-48.478,179.814,6.191,149.173
C02438=1149.039,8.872,-48.465,179.812,6.191,149.173
C02439=1149.044,8.622,-48.450,179.809,6.190,149.174
C02440=1149.049,8.373,-48.437,179.807,6.189,149.174
C02441=1149.054,8.123,-48.423,179.803,6.188,149.175
C02442=1149.059,7.874,-48.410,179.801,6.187,149.176
C02443=1149.064,7.624,-48.397,179.799,6.186,149.176
C02444=1149.069,7.374,-48.382,179.796,6.186,149.177
C02445=1149.075,7.125,-48.369,179.794,6.184,149.177
C02446=1149.079,6.875,-48.355,179.791,6.184,149.178
C02447=1149.085,6.625,-48.342,179.789,6.183,149.178
C02448=1149.090,6.376,-48.328,179.786,6.183,149.179
C02449=1149.095,6.126,-48.315,179.784,6.182,149.179
C02450=1149.100,5.877,-48.301,179.781,6.181,149.180
C02451=1149.106,5.627,-48.288,179.779,6.180,149.181
C02452=1149.110,5.378,-48.274,179.776,6.179,149.181
C02453=1149.116,5.128,-48.261,179.774,6.179,149.182
C02454=1149.120,4.879,-48.247,179.771,6.178,149.182
C02455=1149.126,4.629,-48.234,179.769,6.177,149.183
C02456=1149.131,4.379,-48.220,179.766,6.176,149.183
C02457=1149.136,4.130,-48.207,179.764,6.175,149.184
C02458=1149.141,3.880,-48.193,179.761,6.174,149.185
C02459=1149.146,3.631,-48.180,179.759,6.174,149.185
C02460=1149.151,3.381,-48.167,179.757,6.173,149.186
C02461=1149.156,3.132,-48.153,179.754,6.173,149.186
C02462=1149.161,2.882,-48.140,179.751,6.171,149.187
C02463=1149.167,2.632,-48.127,179.748,6.171,149.187
C02464=1149.171,2.383,-48.113,179.746,6.170,149.188
C02465=1149.177,2.133,-48.100,179.744,6.169,149.189
C02466=1149.182,1.864,-48.085,179.741,6.169,149.189
C02467=1149.188,1.594,-48.071,179.738,6.167,149.190
C02468=1149.194,1.325,-48.057,179.736,6.167,149.190
C02469=1149.199,1.055,-48.043,179.733,6.166,149.191
C02470=1149.204,0.806,-48.029,179.730,6.165,149.192
C02471=1149.209,0.556,-48.016,179.728,6.164,149.192
C02472=1149.215,0.307,-48.003,179.725,6.164,149.193
C02473=1149.219,0.057,-47.989,179.723,6.163,149.193
C02474=1149.225,-0.192,-47.976,179.721,6.162,149.194
C02475=1149.229,-0.442,-47.963,179.718,6.162,149.194
C02476=1149.235,-0.692,-47.950,179.715,6.160,149.195
C02477=1149.239,-0.941,-47.936,179.713,6.160,149.196
C02478=1149.245,-1.191,-47.923,179.711,6.159,149.196
C02479=1149.250,-1.440,-47.910,179.708,6.158,149.197
C02480=1149.256,-1.691,-47.897,179.706,6.157,149.197
C02481=1149.261,-1.940,-47.884,179.703,6.157,149.198
C02482=1149.266,-2.190,-47.870,179.701,6.156,149.198
C02483=1149.271,-2.439,-47.857,179.698,6.155,149.199
C02484=1149.276,-2.688,-47.845,179.696,6.154,149.199
C02485=1149.281,-2.939,-47.831,179.693,6.153,149.200
C02486=1149.286,-3.188,-47.818,179.691,6.153,149.201
C02487=1149.291,-3.438,-47.804,179.689,6.152,149.201
C02488=1149.296,-3.687,-47.792,179.686,6.152,149.202
C02489=1149.302,-3.936,-47.779,179.684,6.151,149.202
C02490=1149.307,-4.187,-47.765,179.681,6.150,149.203
C02491=1149.312,-4.436,-47.753,179.678,6.149,149.203
C02492=1149.318,-4.686,-47.740,179.676,6.148,149.204
C02493=1149.322,-4.936,-47.727,179.673,6.148,149.205
C02494=1149.327,-5.184,-47.713,179.671,6.147,149.205
C02495=1149.333,-5.434,-47.700,179.669,6.146,149.206
C02496=1149.338,-5.684,-47.687,179.666,6.146,149.206
C02497=1149.343,-5.933,-47.675,179.664,6.145,149.207
C02498=1149.349,-6.183,-47.661,179.662,6.144,149.207
C02499=1149.353,-6.433,-47.648,179.658,6.143,149.208
C02500=1149.358,-6.682,-47.636,179.656,6.142,149.209
C02501=1149.364,-6.932,-47.623,179.654,6.142,149.209
C02502=1149.369,-7.182,-47.610,179.651,6.141,149.210
C02503=1149.374,-7.431,-47.597,179.649,6.141,149.210
C02504=1149.380,-7.681,-47.584,179.647,6.140,149.211
C02505=1149.384,-7.931,-47.571,179.644,6.139,149.212
C02506=1149.389,-8.180,-47.558,179.642,6.139,149.212
C02507=1149.394,-8.429,-47.546,179.639,6.138,149.213
C02508=1149.400,-8.680,-47.532,179.636,6.137,149.213
C02509=1149.405,-8.929,-47.520,179.634,6.136,149.214
C02510=1149.410,-9.178,-47.507,179.631,6.135,149.214
C02511=1149.415,-9.428,-47.494,179.629,6.134,149.215
C02512=1149.420,-9.678,-47.481,179.627,6.134,149.215
C02513=1149.425,-9.927,-47.468,179.624,6.133,149.216
C02514=1149.430,-10.177,-47.456,179.622,6.133,149.217
C02515=1149.435,-10.427,-47.443,179.620,6.132,149.217
C02516=1149.441,-10.676,-47.429,179.617,6.132,149.218
C02517=1149.446,-10.926,-47.417,179.615,6.131,149.218
C02518=1149.451,-11.175,-47.404,179.612,6.130,149.219
C02519=1149.456,-11.425,-47.391,179.609,6.129,149.219
C02520=1149.461,-11.674,-47.379,179.607,6.128,149.220
C02521=1149.467,-11.925,-47.366,179.604,6.128,149.221
C02522=1149.472,-12.174,-47.354,179.602,6.127,149.221
C02523=1149.477,-12.424,-47.341,179.600,6.126,149.222
C02524=1149.482,-12.673,-47.328,179.597,6.125,149.222
C02525=1149.487,-12.922,-47.315,179.595,6.125,149.223
C02526=1149.493,-13.172,-47.302,179.593,6.124,149.223
C02527=1149.498,-13.421,-47.290,179.590,6.124,149.224
C02528=1149.503,-13.672,-47.277,179.588,6.123,149.225
C02529=1149.508,-13.921,-47.265,179.585,6.123,149.225
C02530=1149.513,-14.171,-47.252,179.583,6.122,149.226
C02531=1149.518,-14.420,-47.240,179.580,6.121,149.226
C02532=1149.523,-14.669,-47.227,179.578,6.121,149.227
C02533=1149.529,-14.920,-47.214,179.575,6.119,149.228
C02534=1149.534,-15.170,-47.201,179.573,6.119,149.228
C02535=1149.539,-15.419,-47.189,179.570,6.118,149.228
C02536=1149.544,-15.668,-47.176,179.568,6.117,149.229
C02537=1149.549,-15.918,-47.164,179.566,6.116,149.230
C02538=1149.554,-16.168,-47.151,179.563,6.116,149.230
C02539=1149.559,-16.418,-47.139,179.561,6.115,149.231
C02540=1149.564,-16.667,-47.126,179.558,6.115,149.232
C02541=1149.570,-16.917,-47.114,179.556,6.114,149.232
C02542=1149.576,-17.166,-47.101,179.553,6.114,149.233
C02543=1149.581,-17.416,-47.089,179.551,6.113,149.233
C02544=1149.585,-17.666,-47.076,179.548,6.112,149.234
C02545=1149.591,-17.916,-47.064,179.546,6.112,149.234
C02546=1149.596,-18.165,-47.051,179.544,6.111,149.235
C02547=1149.601,-18.415,-47.039,179.541,6.110,149.235
C02548=1149.606,-18.664,-47.027,179.539,6.110,149.236
C02549=1149.611,-18.914,-47.014,179.537,6.109,149.237
C02550=1149.617,-19.164,-47.002,179.534,6.108,149.237
C02551=1149.621,-19.414,-46.989,179.532,6.108,149.238
C02552=1149.626,-19.663,-46.977,179.530,6.107,149.238
C02553=1149.632,-19.913,-46.965,179.527,6.107,149.239
C02554=1149.637,-20.162,-46.952,179.525,6.106,149.239
C02555=1149.642,-20.411,-46.939,179.521,6.105,149.240
C02556=1149.648,-20.661,-46.928,179.519,6.104,149.241
C02557=1149.653,-20.911,-46.915,179.517,6.103,149.241
C02558=1149.658,-21.161,-46.903,179.514,6.103,149.242
C02559=1149.663,-21.410,-46.890,179.512,6.102,149.242
C02560=1149.669,-21.660,-46.879,179.510,6.101,149.243
C02561=1149.673,-21.910,-46.866,179.507,6.101,149.243
C02562=1149.678,-22.159,-46.853,179.505,6.100,149.244
C02563=1149.684,-22.409,-46.841,179.503,6.099,149.245
C02564=1149.689,-22.658,-46.829,179.500,6.099,149.245
C02565=1149.694,-22.908,-46.817,179.498,6.098,149.246
C02566=1149.699,-23.158,-46.804,179.495,6.098,149.246
C02567=1149.705,-23.408,-46.792,179.493,6.097,149.247
C02568=1149.710,-23.657,-46.780,179.491,6.096,149.247
C02569=1149.715,-23.907,-46.768,179.488,6.096,149.248
C02570=1149.721,-24.177,-46.755,179.485,6.095,149.249
C02571=1149.726,-24.446,-46.741,179.483,6.095,149.249
C02572=1149.732,-24.717,-46.728,179.481,6.094,149.250
C02573=1149.738,-24.987,-46.715,179.478,6.093,149.250
C02574=1149.742,-25.236,-46.703,179.476,6.093,149.251
C02575=1149.748,-25.486,-46.691,179.474,6.092,149.252
C02576=1149.753,-25.736,-46.678,179.471,6.092,149.252
C02577=1149.758,-25.985,-46.667,179.469,6.091,149.253
C02578=1149.763,-26.235,-46.655,179.466,6.090,149.253
C02579=1149.769,-26.485,-46.642,179.464,6.090,149.254
C02580=1149.774,-26.735,-46.630,179.461,6.089,149.255
C02581=1149.778,-26.984,-46.618,179.459,6.088,149.255
C02582=1149.784,-27.234,-46.606,179.456,6.088,149.256
C02583=1149.789,-27.484,-46.594,179.454,6.087,149.256
C02584=1149.794,-27.733,-46.582,179.452,6.086,149.257
C02585=1149.800,-27.983,-46.570,179.449,6.086,149.257
C02586=1149.805,-28.233,-46.558,179.447,6.085,149.258
C02587=1149.810,-28.482,-46.546,179.444,6.085,149.259
C02588=1149.815,-28.732,-46.534,179.442,6.084,149.259
C02589=1149.821,-28.982,-46.522,179.440,6.084,149.260
C02590=1149.826,-29.231,-46.510,179.437,6.083,149.260
C02591=1149.831,-29.481,-46.498,179.435,6.082,149.261
C02592=1149.836,-29.731,-46.486,179.433,6.082,149.261
C02593=1149.841,-29.980,-46.474,179.430,6.081,149.262
C02594=1149.846,-30.230,-46.462,179.428,6.080,149.263
C02595=1149.852,-30.480,-46.450,179.426,6.080,149.263
C02596=1149.857,-30.728,-46.438,179.423,6.079,149.264
C02597=1149.862,-30.978,-46.427,179.421,6.078,149.264
C02598=1149.868,-31.228,-46.415,179.418,6.078,149.265
C02599=1149.873,-31.478,-46.403,179.416,6.077,149.265
C02600=1149.877,-31.727,-46.391,179.413,6.077,149.266
C02601=1149.883,-31.977,-46.379,179.411,6.076,149.267
C02602=1149.888,-32.227,-46.367,179.409,6.075,149.267
C02603=1149.894,-32.477,-46.355,179.406,6.075,149.268
C02604=1149.898,-32.726,-46.344,179.404,6.074,149.268
C02605=1149.904,-32.976,-46.331,179.401,6.074,149.269
C02606=1149.909,-33.226,-46.319,179.399,6.073,149.269
C02607=1149.914,-33.475,-46.307,179.396,6.072,149.270
C02608=1149.919,-33.725,-46.296,179.394,6.072,149.271
C02609=1149.925,-33.974,-46.285,179.392,6.071,149.271
C02610=1149.930,-34.224,-46.272,179.389,6.070,149.272
C02611=1149.935,-34.473,-46.261,179.387,6.070,149.272
C02612=1149.940,-34.723,-46.249,179.385,6.070,149.273
C02613=1149.946,-34.973,-46.237,179.383,6.069,149.273
C02614=1149.950,-35.223,-46.226,179.380,6.069,149.274
C02615=1149.956,-35.473,-46.214,179.378,6.068,149.275
C02616=1149.961,-35.723,-46.202,179.375,6.068,149.275
C02617=1149.966,-35.972,-46.191,179.373,6.067,149.276
C02618=1149.972,-36.221,-46.178,179.371,6.066,149.276
C02619=1149.977,-36.471,-46.167,179.368,6.066,149.277
C02620=1149.982,-36.720,-46.155,179.366,6.065,149.277
C02621=1149.987,-36.970,-46.143,179.364,6.064,149.278
C02622=1149.993,-37.220,-46.131,179.361,6.064,149.279
C02623=1149.997,-37.470,-46.120,179.359,6.063,149.279
C02624=1150.003,-37.720,-46.108,179.357,6.062,149.280
C02625=1150.008,-37.969,-46.097,179.354,6.062,149.280
C02626=1150.014,-38.219,-46.085,179.352,6.061,149.281
C02627=1150.019,-38.469,-46.074,179.350,6.061,149.281
C02628=1150.024,-38.718,-46.062,179.347,6.061,149.282
C02629=1150.029,-38.968,-46.050,179.345,6.060,149.283
C02630=1150.034,-39.217,-46.039,179.343,6.060,149.283
C02631=1150.040,-39.467,-46.028,179.340,6.059,149.284
C02632=1150.045,-39.717,-46.016,179.338,6.058,149.284
C02633=1150.050,-39.967,-46.004,179.336,6.058,149.285
C02634=1150.055,-40.217,-45.993,179.333,6.057,149.285
C02635=1150.060,-40.466,-45.981,179.331,6.056,149.286
C02636=1150.066,-40.715,-45.970,179.329,6.056,149.287
C02637=1150.071,-40.965,-45.958,179.326,6.055,149.287
C02638=1150.076,-41.215,-45.947,179.324,6.054,149.288
C02639=1150.081,-41.465,-45.935,179.322,6.054,149.288
C02640=1150.087,-41.714,-45.924,179.319,6.054,149.289
C02641=1150.092,-41.963,-45.912,179.317,6.053,149.289
C02642=1150.097,-42.213,-45.901,179.315,6.053,149.290
C02643=1150.102,-42.463,-45.889,179.312,6.052,149.291
C02644=1150.107,-42.714,-45.878,179.310,6.052,149.291
C02645=1150.113,-42.963,-45.867,179.308,6.051,149.292
C02646=1150.118,-43.212,-45.855,179.305,6.050,149.292
C02647=1150.123,-43.462,-45.844,179.303,6.050,149.293
C02648=1150.128,-43.712,-45.832,179.301,6.049,149.293
C02649=1150.134,-43.961,-45.821,179.298,6.049,149.294
C02650=1150.139,-44.211,-45.809,179.296,6.048,149.295
C02651=1150.144,-44.461,-45.799,179.294,6.048,149.295
C02652=1150.149,-44.711,-45.787,179.291,6.047,149.296
C02653=1150.155,-44.960,-45.776,179.289,6.046,149.296
C02654=1150.160,-45.210,-45.764,179.287,6.046,149.297
C02655=1150.165,-45.460,-45.753,179.284,6.045,149.297
C02656=1150.170,-45.709,-45.741,179.282,6.045,149.298
C02657=1150.176,-45.959,-45.731,179.280,6.044,149.299
C02658=1150.181,-46.209,-45.719,179.277,6.044,149.299
C02659=1150.186,-46.459,-45.707,179.275,6.044,149.300
C02660=1150.191,-46.708,-45.697,179.273,6.043,149.300
C02661=1150.197,-46.957,-45.685,179.270,6.042,149.301
C02662=1150.202,-47.208,-45.674,179.268,6.042,149.301
C02663=1150.206,-47.457,-45.663,179.266,6.041,149.302
C02664=1150.212,-47.707,-45.651,179.263,6.040,149.303
C02665=1150.217,-47.956,-45.640,179.261,6.040,149.303
C02666=1150.223,-48.207,-45.629,179.259,6.040,149.304
C02667=1150.228,-48.456,-45.618,179.257,6.039,149.304
C02668=1150.233,-48.705,-45.607,179.254,6.039,149.305
C02669=1150.239,-48.956,-45.595,179.252,6.038,149.305
C02670=1150.244,-49.205,-45.585,179.249,6.038,149.306
C02671=1150.249,-49.454,-45.573,179.247,6.037,149.307
C02672=1150.254,-49.705,-45.562,179.245,6.036,149.307
C02673=1150.260,-49.954,-45.551,179.242,6.036,149.308
C02674=1150.265,-50.225,-45.539,179.240,6.035,149.308
C02675=1150.271,-50.496,-45.527,179.238,6.035,149.309
C02676=1150.277,-50.766,-45.515,179.235,6.034,149.310
C02677=1150.282,-51.037,-45.503,179.233,6.033,149.310
C02678=1150.288,-51.286,-45.492,179.231,6.034,149.311
C02679=1150.293,-51.536,-45.480,179.228,6.033,149.311
C02680=1150.298,-51.786,-45.470,179.226,6.032,149.312
C02681=1150.304,-52.035,-45.458,179.224,6.032,149.313
C02682=1150.309,-52.285,-45.448,179.221,6.031,149.313
C02683=1150.313,-52.535,-45.436,179.219,6.031,149.314
C02684=1150.319,-52.784,-45.425,179.216,6.030,149.314
C02685=1150.324,-53.034,-45.414,179.215,6.030,149.315
C02686=1150.329,-53.284,-45.403,179.212,6.029,149.315
C02687=1150.335,-53.534,-45.393,179.210,6.029,149.316
C02688=1150.339,-53.783,-45.381,179.207,6.028,149.317
C02689=1150.346,-54.033,-45.371,179.205,6.028,149.317
C02690=1150.350,-54.283,-45.359,179.203,6.027,149.317
C02691=1150.355,-54.532,-45.348,179.201,6.027,149.318
C02692=1150.361,-54.782,-45.338,179.199,6.026,149.319
C02693=1150.366,-55.032,-45.326,179.196,6.026,149.319
C02694=1150.372,-55.281,-45.316,179.194,6.025,149.320
C02695=1150.376,-55.531,-45.304,179.192,6.024,149.320
C02696=1150.381,-55.781,-45.294,179.189,6.024,149.321
C02697=1150.387,-56.030,-45.283,179.187,6.024,149.322
C02698=1150.392,-56.281,-45.272,179.185,6.024,149.322
C02699=1150.398,-56.530,-45.261,179.183,6.023,149.323
C02700=1150.403,-56.780,-45.250,179.180,6.022,149.323
C02701=1150.408,-57.029,-45.239,179.178,6.022,149.324
C02702=1150.413,-57.279,-45.229,179.176,6.021,149.324
C02703=1150.419,-57.529,-45.217,179.173,6.021,149.325
C02704=1150.424,-57.779,-45.207,179.171,6.020,149.326
C02705=1150.429,-58.029,-45.196,179.169,6.020,149.326
C02706=1150.434,-58.278,-45.185,179.166,6.019,149.327
C02707=1150.439,-58.528,-45.175,179.164,6.019,149.327
C02708=1150.445,-58.777,-45.164,179.162,6.018,149.328
C02709=1150.450,-59.027,-45.153,179.160,6.018,149.328
C02710=1150.456,-59.276,-45.142,179.158,6.017,149.329
C02711=1150.461,-59.527,-45.131,179.155,6.017,149.330
C02712=1150.466,-59.776,-45.121,179.153,6.016,149.330
C02713=1150.471,-60.026,-45.110,179.150,6.016,149.331
C02714=1150.477,-60.275,-45.099,179.149,6.016,149.331
C02715=1150.482,-60.526,-45.089,179.146,6.015,149.332
C02716=1150.486,-60.775,-45.077,179.144,6.015,149.332
C02717=1150.492,-61.025,-45.067,179.142,6.014,149.333
C02718=1150.498,-61.275,-45.056,179.139,6.013,149.333
C02719=1150.503,-61.524,-45.045,179.137,6.013,149.334
C02720=1150.508,-61.774,-45.035,179.135,6.013,149.335
C02721=1150.514,-62.024,-45.024,179.133,6.012,149.335
C02722=1150.518,-62.274,-45.013,179.130,6.012,149.336
C02723=1150.524,-62.523,-45.003,179.128,6.011,149.336
C02724=1150.529,-62.773,-44.993,179.126,6.011,149.337
C02725=1150.534,-63.022,-44.981,179.124,6.010,149.337
C02726=1150.540,-63.272,-44.971,179.121,6.010,149.338
C02727=1150.545,-63.522,-44.961,179.119,6.009,149.339
C02728=1150.550,-63.772,-44.950,179.117,6.008,149.339
C02729=1150.555,-64.021,-44.939,179.115,6.009,149.340
C02730=1150.561,-64.271,-44.929,179.113,6.008,149.340
C02731=1150.566,-64.521,-44.918,179.110,6.007,149.341
C02732=1150.571,-64.771,-44.908,179.108,6.007,149.341
C02733=1150.576,-65.020,-44.897,179.106,6.007,149.342
C02734=1150.581,-65.270,-44.887,179.103,6.007,149.343
C02735=1150.586,-65.520,-44.876,179.101,6.006,149.343
C02736=1150.592,-65.770,-44.866,179.099,6.005,149.344
C02737=1150.597,-66.019,-44.855,179.096,6.005,149.344
C02738=1150.602,-66.269,-44.844,179.095,6.005,149.345
C02739=1150.608,-66.518,-44.834,179.093,6.004,149.345
C02740=1150.613,-66.769,-44.824,179.090,6.003,149.346
C02741=1150.619,-67.018,-44.813,179.088,6.003,149.346
C02742=1150.624,-67.268,-44.803,179.086,6.003,149.347
C02743=1150.629,-67.517,-44.792,179.083,6.002,149.348
C02744=1150.634,-67.767,-44.782,179.081,6.002,149.348
C02745=1150.639,-68.017,-44.771,179.079,6.001,149.349
C02746=1150.645,-68.267,-44.761,179.076,6.000,149.349
C02747=1150.650,-68.517,-44.750,179.075,6.000,149.350
C02748=1150.656,-68.766,-44.740,179.072,6.000,149.351
C02749=1150.661,-69.016,-44.730,179.070,5.999,149.351
C02750=1150.666,-69.266,-44.719,179.068,5.998,149.351
C02751=1150.672,-69.515,-44.708,179.066,5.999,149.352
C02752=1150.677,-69.765,-44.698,179.064,5.998,149.353
C02753=1150.682,-70.015,-44.688,179.061,5.997,149.353
C02754=1150.688,-70.264,-44.677,179.059,5.997,149.354
C02755=1150.693,-70.515,-44.667,179.057,5.997,149.354
C02756=1150.698,-70.764,-44.657,179.054,5.997,149.355
C02757=1150.703,-71.013,-44.647,179.052,5.996,149.356
C02758=1150.708,-71.264,-44.636,179.050,5.995,149.356
C02759=1150.714,-71.513,-44.626,179.048,5.995,149.357
C02760=1150.719,-71.763,-44.616,179.046,5.995,149.357
C02761=1150.724,-72.013,-44.605,179.044,5.994,149.358
C02762=1150.730,-72.263,-44.595,179.041,5.993,149.358
C02763=1150.736,-72.512,-44.585,179.039,5.993,149.359
C02764=1150.741,-72.762,-44.574,179.037,5.993,149.359
C02765=1150.745,-73.012,-44.565,179.034,5.992,149.360
C02766=1150.751,-73.261,-44.555,179.032,5.992,149.361
C02767=1150.756,-73.511,-44.544,179.031,5.992,149.361
C02768=1150.762,-73.761,-44.534,179.028,5.991,149.362
C02769=1150.767,-74.010,-44.524,179.026,5.990,149.362
C02770=1150.772,-74.261,-44.513,179.024,5.990,149.363
C02771=1150.778,-74.510,-44.503,179.022,5.990,149.363
C02772=1150.783,-74.759,-44.493,179.019,5.989,149.364
C02773=1150.788,-75.010,-44.483,179.017,5.988,149.364
C02774=1150.793,-75.259,-44.472,179.015,5.989,149.365
C02775=1150.799,-75.509,-44.462,179.013,5.988,149.366
C02776=1150.804,-75.758,-44.452,179.011,5.987,149.366
C02777=1150.809,-76.008,-44.442,179.008,5.987,149.367
C02778=1150.815,-76.279,-44.431,179.006,5.986,149.367
C02779=1150.821,-76.551,-44.421,179.004,5.987,149.368
C02780=1150.827,-76.823,-44.409,179.002,5.986,149.368
C02781=1150.832,-77.093,-44.399,178.999,5.985,149.369
C02782=1150.837,-77.344,-44.388,178.997,5.985,149.370
C02783=1150.843,-77.593,-44.378,178.994,5.984,149.370
C02784=1150.849,-77.843,-44.368,178.992,5.984,149.371
C02785=1150.853,-78.093,-44.358,178.990,5.984,149.371
C02786=1150.859,-78.343,-44.348,178.988,5.983,149.372
C02787=1150.864,-78.592,-44.338,178.986,5.983,149.372
C02788=1150.870,-78.842,-44.328,178.984,5.982,149.373
C02789=1150.874,-79.092,-44.318,178.981,5.982,149.374
C02790=1150.880,-79.341,-44.307,178.979,5.981,149.374
C02791=1150.886,-79.591,-44.298,178.977,5.981,149.375
C02792=1150.891,-79.841,-44.288,178.975,5.981,149.375
C02793=1150.896,-80.091,-44.278,178.972,5.980,149.376
C02794=1150.901,-80.341,-44.268,178.971,5.980,149.376
C02795=1150.907,-80.590,-44.257,178.968,5.980,149.377
C02796=1150.912,-80.840,-44.248,178.966,5.979,149.377
C02797=1150.918,-81.089,-44.238,178.964,5.978,149.378
C02798=1150.923,-81.340,-44.228,178.962,5.979,149.379
C02799=1150.927,-81.589,-44.218,178.960,5.978,149.379
C02800=1150.933,-81.838,-44.208,178.957,5.977,149.380
C02801=1150.939,-82.089,-44.198,178.955,5.978,149.380
C02802=1150.944,-82.339,-44.188,178.953,5.977,149.381
C02803=1150.949,-82.588,-44.178,178.951,5.976,149.381
C02804=1150.955,-82.838,-44.169,178.949,5.976,149.382
C02805=1150.960,-83.088,-44.158,178.947,5.976,149.383
C02806=1150.965,-83.337,-44.149,178.944,5.975,149.383
C02807=1150.971,-83.587,-44.139,178.943,5.975,149.383
C02808=1150.975,-83.837,-44.129,178.940,5.975,149.384
C02809=1150.981,-84.087,-44.119,178.938,5.974,149.385
C02810=1150.987,-84.336,-44.109,178.936,5.973,149.385
C02811=1150.992,-84.586,-44.100,178.934,5.973,149.386
C02812=1150.997,-84.836,-44.090,178.931,5.973,149.386
C02813=1151.002,-85.086,-44.079,178.929,5.972,149.387
C02814=1151.007,-85.336,-44.070,178.927,5.972,149.388
C02815=1151.013,-85.585,-44.060,178.925,5.972,149.388
C02816=1151.018,-85.834,-44.051,178.923,5.971,149.389
C02817=1151.024,-86.085,-44.041,178.921,5.971,149.389
C02818=1151.029,-86.334,-44.031,178.919,5.970,149.390
C02819=1151.034,-86.584,-44.021,178.916,5.970,149.390
C02820=1151.040,-86.834,-44.011,178.915,5.970,149.391
C02821=1151.044,-87.084,-44.002,178.912,5.969,149.391
C02822=1151.050,-87.334,-43.992,178.910,5.969,149.392
C02823=1151.055,-87.583,-43.983,178.908,5.969,149.392
C02824=1151.061,-87.832,-43.972,178.906,5.968,149.393
C02825=1151.066,-88.082,-43.964,178.903,5.967,149.394
C02826=1151.071,-88.333,-43.953,178.902,5.967,149.394
C02827=1151.076,-88.582,-43.944,178.900,5.967,149.395
C02828=1151.082,-88.832,-43.934,178.897,5.966,149.395
C02829=1151.088,-89.082,-43.924,178.895,5.966,149.396
C02830=1151.092,-89.331,-43.915,178.893,5.966,149.396
C02831=1151.098,-89.582,-43.905,178.891,5.965,149.397
C02832=1151.103,-89.831,-43.896,178.889,5.965,149.397
C02833=1151.109,-90.080,-43.885,178.887,5.964,149.398
C02834=1151.114,-90.330,-43.877,178.885,5.964,149.398
C02835=1151.119,-90.580,-43.866,178.882,5.964,149.399
C02836=1151.124,-90.830,-43.857,178.880,5.963,149.400
C02837=1151.130,-91.080,-43.847,178.878,5.963,149.400
C02838=1151.135,-91.330,-43.838,178.876,5.963,149.401
C02839=1151.141,-91.579,-43.828,178.874,5.962,149.401
C02840=1151.146,-91.829,-43.819,178.872,5.961,149.402
C02841=1151.151,-92.079,-43.809,178.870,5.962,149.402
C02842=1151.156,-92.328,-43.800,178.867,5.961,149.403
C02843=1151.162,-92.578,-43.791,178.865,5.960,149.403
C02844=1151.167,-92.828,-43.781,178.864,5.960,149.404
C02845=1151.172,-93.078,-43.772,178.861,5.960,149.405
C02846=1151.178,-93.327,-43.762,178.859,5.960,149.405
C02847=1151.183,-93.577,-43.753,178.857,5.959,149.406
C02848=1151.188,-93.827,-43.742,178.855,5.959,149.406
C02849=1151.193,-94.077,-43.733,178.853,5.959,149.407
C02850=1151.199,-94.327,-43.724,178.851,5.958,149.407
C02851=1151.204,-94.577,-43.714,178.848,5.957,149.408
C02852=1151.209,-94.826,-43.705,178.847,5.957,149.408
C02853=1151.215,-95.076,-43.695,178.844,5.957,149.409
C02854=1151.220,-95.326,-43.686,178.842,5.956,149.409
C02855=1151.226,-95.576,-43.677,178.840,5.956,149.410
C02856=1151.231,-95.825,-43.667,178.838,5.956,149.410
C02857=1151.237,-96.075,-43.657,178.836,5.956,149.411
C02858=1151.242,-96.325,-43.648,178.834,5.955,149.412
C02859=1151.247,-96.574,-43.639,178.832,5.954,149.412
C02860=1151.253,-96.825,-43.629,178.830,5.955,149.413
C02861=1151.257,-97.074,-43.620,178.827,5.954,149.413
C02862=1151.263,-97.324,-43.611,178.825,5.953,149.414
C02863=1151.269,-97.574,-43.601,178.824,5.953,149.414
C02864=1151.273,-97.823,-43.592,178.821,5.953,149.415
C02865=1151.279,-98.073,-43.582,178.819,5.952,149.415
C02866=1151.284,-98.323,-43.573,178.817,5.952,149.416
C02867=1151.290,-98.573,-43.565,178.815,5.952,149.416
C02868=1151.295,-98.822,-43.554,178.813,5.952,149.417
C02869=1151.300,-99.072,-43.545,178.811,5.951,149.418
C02870=1151.306,-99.322,-43.537,178.809,5.950,149.418
C02871=1151.311,-99.572,-43.526,178.807,5.950,149.419
C02872=1151.316,-99.822,-43.517,178.804,5.950,149.419
C02873=1151.322,-100.071,-43.509,178.803,5.950,149.420
C02874=1151.327,-100.322,-43.499,178.800,5.949,149.420
C02875=1151.332,-100.571,-43.489,178.798,5.949,149.421
C02876=1151.337,-100.821,-43.481,178.796,5.949,149.421
C02877=1151.343,-101.071,-43.471,178.794,5.948,149.422
C02878=1151.349,-101.321,-43.462,178.792,5.948,149.422
C02879=1151.353,-101.570,-43.453,178.790,5.948,149.423
C02880=1151.359,-101.819,-43.444,178.788,5.947,149.423
C02881=1151.365,-102.069,-43.435,178.786,5.947,149.424
C02882=1151.371,-102.341,-43.424,178.784,5.946,149.425
C02883=1151.376,-102.614,-43.415,178.781,5.946,149.425
C02884=1151.382,-102.886,-43.405,178.779,5.945,149.426
C02885=1151.387,-103.158,-43.394,178.777,5.945,149.426
C02886=1151.393,-103.407,-43.385,178.775,5.945,149.427
C02887=1151.398,-103.658,-43.376,178.773,5.945,149.427
C02888=1151.404,-103.907,-43.367,178.771,5.944,149.428
C02889=1151.409,-104.157,-43.359,178.769,5.944,149.428
C02890=1151.415,-104.406,-43.350,178.767,5.944,149.429
C02891=1151.420,-104.657,-43.340,178.764,5.943,149.430
C02892=1151.425,-104.906,-43.331,178.763,5.943,149.430
C02893=1151.430,-105.156,-43.322,178.761,5.942,149.431
C02894=1151.436,-105.406,-43.313,178.758,5.942,149.431
C02895=1151.442,-105.656,-43.303,178.756,5.942,149.432
C02896=1151.447,-105.906,-43.294,178.754,5.941,149.432
C02897=1151.452,-106.155,-43.285,178.752,5.941,149.433
C02898=1151.457,-106.405,-43.277,178.750,5.941,149.433
C02899=1151.462,-106.655,-43.268,178.748,5.940,149.434
C02900=1151.469,-106.905,-43.258,178.746,5.940,149.434
C02901=1151.474,-107.154,-43.249,178.744,5.940,149.435
C02902=1151.479,-107.404,-43.240,178.742,5.940,149.435
C02903=1151.484,-107.653,-43.231,178.740,5.939,149.436
C02904=1151.489,-107.903,-43.222,178.738,5.939,149.437
C02905=1151.494,-108.153,-43.213,178.736,5.939,149.437
C02906=1151.500,-108.403,-43.204,178.734,5.938,149.438
C02907=1151.506,-108.652,-43.195,178.732,5.938,149.438
C02908=1151.511,-108.902,-43.186,178.730,5.937,149.439
C02909=1151.516,-109.152,-43.177,178.728,5.937,149.439
C02910=1151.521,-109.402,-43.169,178.725,5.937,149.440
C02911=1151.527,-109.652,-43.160,178.723,5.936,149.440
C02912=1151.532,-109.902,-43.151,178.722,5.936,149.441
C02913=1151.538,-110.152,-43.141,178.720,5.935,149.441
C02914=1151.543,-110.401,-43.133,178.717,5.936,149.442
C02915=1151.549,-110.651,-43.124,178.715,5.935,149.442
C02916=1151.554,-110.901,-43.115,178.714,5.935,149.443
C02917=1151.559,-111.151,-43.106,178.711,5.934,149.443
C02918=1151.564,-111.400,-43.097,178.710,5.934,149.444
C02919=1151.569,-111.650,-43.088,178.707,5.934,149.445
C02920=1151.575,-111.899,-43.080,178.705,5.933,149.445
C02921=1151.580,-112.149,-43.071,178.703,5.933,149.446
C02922=1151.586,-112.399,-43.061,178.701,5.932,149.446
C02923=1151.591,-112.649,-43.052,178.700,5.932,149.447
C02924=1151.597,-112.900,-43.044,178.697,5.932,149.447
C02925=1151.602,-113.149,-43.036,178.695,5.932,149.448
C02926=1151.608,-113.399,-43.027,178.693,5.931,149.448
C02927=1151.613,-113.649,-43.018,178.691,5.931,149.449
C02928=1151.618,-113.899,-43.009,178.689,5.931,149.449
C02929=1151.623,-114.148,-43.000,178.687,5.930,149.450
C02930=1151.629,-114.397,-42.992,178.685,5.930,149.450
C02931=1151.634,-114.647,-42.983,178.683,5.930,149.451
C02932=1151.639,-114.897,-42.974,178.681,5.930,149.451
C02933=1151.645,-115.148,-42.966,178.679,5.929,149.452
C02934=1151.650,-115.397,-42.957,178.677,5.929,149.452
C02935=1151.656,-115.647,-42.948,178.675,5.928,149.453
C02936=1151.661,-115.897,-42.939,178.673,5.929,149.454
C02937=1151.666,-116.146,-42.930,178.671,5.928,149.454
C02938=1151.671,-116.396,-42.922,178.669,5.927,149.455
C02939=1151.677,-116.645,-42.913,178.667,5.927,149.455
C02940=1151.682,-116.896,-42.905,178.665,5.926,149.456
C02941=1151.688,-117.146,-42.896,178.663,5.926,149.456
C02942=1151.693,-117.396,-42.887,178.661,5.926,149.456
C02943=1151.698,-117.645,-42.878,178.659,5.926,149.457
C02944=1151.704,-117.895,-42.870,178.657,5.925,149.458
C02945=1151.709,-118.145,-42.861,178.655,5.925,149.458
C02946=1151.714,-118.395,-42.852,178.653,5.925,149.459
C02947=1151.720,-118.644,-42.844,178.652,5.925,149.459
C02948=1151.725,-118.894,-42.835,178.649,5.924,149.460
C02949=1151.731,-119.144,-42.827,178.647,5.924,149.460
C02950=1151.736,-119.393,-42.818,178.645,5.924,149.461
C02951=1151.742,-119.643,-42.809,178.643,5.923,149.461
C02952=1151.747,-119.893,-42.801,178.641,5.923,149.462
C02953=1151.752,-120.143,-42.792,178.639,5.922,149.462
C02954=1151.758,-120.393,-42.784,178.637,5.922,149.463
C02955=1151.763,-120.643,-42.775,178.635,5.921,149.463
C02956=1151.768,-120.893,-42.766,178.633,5.922,149.464
C02957=1151.774,-121.142,-42.758,178.631,5.921,149.464
C02958=1151.780,-121.392,-42.749,178.629,5.921,149.465
C02959=1151.785,-121.642,-42.740,178.627,5.920,149.465
C02960=1151.790,-121.892,-42.732,178.626,5.920,149.466
C02961=1151.795,-122.141,-42.724,178.623,5.920,149.466
C02962=1151.800,-122.391,-42.715,178.622,5.920,149.467
C02963=1151.806,-122.641,-42.707,178.619,5.919,149.468
C02964=1151.812,-122.891,-42.699,178.618,5.919,149.468
C02965=1151.817,-123.141,-42.690,178.615,5.919,149.469
C02966=1151.822,-123.390,-42.681,178.614,5.919,149.469
C02967=1151.828,-123.640,-42.673,178.612,5.918,149.470
C02968=1151.833,-123.890,-42.664,178.610,5.918,149.470
C02969=1151.838,-124.140,-42.655,178.608,5.917,149.471
C02970=1151.844,-124.389,-42.648,178.606,5.917,149.471
C02971=1151.849,-124.639,-42.639,178.604,5.916,149.472
C02972=1151.854,-124.890,-42.631,178.602,5.917,149.472
C02973=1151.860,-125.139,-42.622,178.600,5.916,149.473
C02974=1151.865,-125.389,-42.614,178.598,5.916,149.473
C02975=1151.871,-125.639,-42.605,178.596,5.915,149.474
C02976=1151.877,-125.888,-42.597,178.594,5.915,149.474
C02977=1151.881,-126.139,-42.589,178.592,5.915,149.475
C02978=1151.886,-126.388,-42.580,178.591,5.915,149.475
C02979=1151.892,-126.638,-42.572,178.588,5.914,149.476
C02980=1151.898,-126.888,-42.564,178.587,5.914,149.476
C02981=1151.903,-127.137,-42.555,178.584,5.914,149.477
C02982=1151.908,-127.387,-42.548,178.582,5.914,149.477
C02983=1151.913,-127.637,-42.539,178.580,5.913,149.478
C02984=1151.919,-127.887,-42.531,178.579,5.913,149.478
C02985=1151.925,-128.137,-42.522,178.576,5.912,149.479
C02986=1151.504,-128.148,-42.565,178.573,5.916,149.481
C02987=1151.498,-127.898,-42.573,178.575,5.916,149.480
C02988=1151.493,-127.648,-42.581,178.576,5.916,149.480
C02989=1151.487,-127.399,-42.590,178.579,5.917,149.479
C02990=1151.482,-127.149,-42.598,178.581,5.917,149.478
C02991=1151.477,-126.899,-42.606,178.583,5.917,149.478
C02992=1151.471,-126.649,-42.614,178.584,5.917,149.477
C02993=1151.466,-126.399,-42.623,178.587,5.918,149.477
C02994=1151.460,-126.149,-42.631,178.588,5.918,149.477
C02995=1151.455,-125.900,-42.639,178.590,5.919,149.476
C02996=1151.450,-125.650,-42.648,178.592,5.919,149.476
C02997=1151.444,-125.400,-42.656,178.594,5.919,149.475
C02998=1151.439,-125.150,-42.665,178.596,5.919,149.475
C02999=1151.433,-124.900,-42.673,178.599,5.920,149.474
C03000=1151.428,-124.651,-42.682,178.601,5.921,149.473
C03001=1151.422,-124.401,-42.691,178.602,5.920,149.473
C03002=1151.418,-124.151,-42.698,178.605,5.921,149.472
C03003=1151.412,-123.902,-42.707,178.606,5.921,149.472
C03004=1151.407,-123.652,-42.716,178.608,5.922,149.471
C03005=1151.401,-123.401,-42.724,178.610,5.922,149.471
C03006=1151.396,-123.152,-42.732,178.612,5.923,149.470
C03007=1151.390,-122.902,-42.741,178.614,5.922,149.470
C03008=1151.385,-122.652,-42.749,178.616,5.923,149.469
C03009=1151.379,-122.403,-42.758,178.618,5.923,149.469
C03010=1151.374,-122.153,-42.767,178.620,5.924,149.468
C03011=1151.369,-121.903,-42.774,178.622,5.924,149.468
C03012=1151.364,-121.653,-42.783,178.624,5.924,149.467
C03013=1151.358,-121.404,-42.792,178.626,5.924,149.467
C03014=1151.353,-121.153,-42.800,178.628,5.925,149.466
C03015=1151.348,-120.903,-42.809,178.630,5.925,149.466
C03016=1151.342,-120.654,-42.817,178.632,5.925,149.465
C03017=1151.337,-120.404,-42.826,178.634,5.925,149.465
C03018=1151.331,-120.154,-42.834,178.636,5.926,149.464
C03019=1151.326,-119.905,-42.843,178.637,5.926,149.464
C03020=1151.320,-119.655,-42.852,178.640,5.927,149.463
C03021=1151.315,-119.405,-42.861,178.641,5.927,149.463
C03022=1151.310,-119.155,-42.869,178.644,5.927,149.462
C03023=1151.304,-118.905,-42.878,178.645,5.927,149.461
C03024=1151.299,-118.656,-42.886,178.648,5.928,149.461
C03025=1151.294,-118.406,-42.895,178.650,5.929,149.460
C03026=1151.288,-118.155,-42.903,178.651,5.929,149.460
C03027=1151.283,-117.906,-42.911,178.654,5.929,149.459
C03028=1151.278,-117.657,-42.920,178.655,5.929,149.459
C03029=1151.273,-117.407,-42.929,178.658,5.930,149.458
C03030=1151.268,-117.157,-42.938,178.660,5.930,149.458
C03031=1151.262,-116.907,-42.946,178.662,5.930,149.457
C03032=1151.256,-116.657,-42.955,178.663,5.930,149.457
C03033=1151.251,-116.407,-42.964,178.666,5.931,149.456
C03034=1151.245,-116.157,-42.973,178.667,5.931,149.456
C03035=1151.240,-115.908,-42.982,178.669,5.932,149.455
C03036=1151.234,-115.658,-42.991,178.672,5.932,149.455
C03037=1151.229,-115.408,-42.999,178.674,5.932,149.454
C03038=1151.224,-115.158,-43.008,178.676,5.933,149.454
C03039=1151.218,-114.909,-43.016,178.677,5.933,149.453
C03040=1151.213,-114.659,-43.025,178.680,5.934,149.453
C03041=1151.208,-114.409,-43.034,178.681,5.934,149.452
C03042=1151.202,-114.159,-43.043,178.684,5.934,149.452
C03043=1151.197,-113.910,-43.051,178.685,5.934,149.451
C03044=1151.191,-113.660,-43.060,178.688,5.935,149.451
C03045=1151.186,-113.410,-43.069,178.689,5.935,149.450
C03046=1151.181,-113.160,-43.077,178.691,5.935,149.450
C03047=1151.176,-112.910,-43.086,178.694,5.936,149.449
C03048=1151.170,-112.661,-43.095,178.696,5.936,149.448
C03049=1151.165,-112.411,-43.104,178.698,5.936,149.448
C03050=1151.160,-112.161,-43.113,178.700,5.936,149.447
C03051=1151.154,-111.911,-43.122,178.702,5.937,149.447
C03052=1151.149,-111.661,-43.131,178.703,5.937,149.446
C03053=1151.143,-111.411,-43.140,178.706,5.937,149.446
C03054=1151.138,-111.162,-43.149,178.708,5.938,149.445
C03055=1151.132,-110.912,-43.157,178.710,5.938,149.445
C03056=1151.127,-110.662,-43.166,178.712,5.939,149.444
C03057=1151.122,-110.413,-43.175,178.714,5.939,149.444
C03058=1151.117,-110.163,-43.184,178.716,5.939,149.443
C03059=1151.112,-109.913,-43.193,178.718,5.939,149.443
C03060=1151.105,-109.663,-43.202,178.720,5.940,149.442
C03061=1151.100,-109.414,-43.211,178.722,5.940,149.442
C03062=1151.095,-109.164,-43.220,178.724,5.941,149.441
C03063=1151.090,-108.914,-43.229,178.727,5.941,149.440
C03064=1151.085,-108.664,-43.238,178.728,5.941,149.440
C03065=1151.079,-108.414,-43.247,178.730,5.942,149.439
C03066=1151.074,-108.165,-43.255,178.732,5.942,149.439
C03067=1151.068,-107.915,-43.265,178.734,5.943,149.438
C03068=1151.063,-107.665,-43.274,178.737,5.943,149.438
C03069=1151.057,-107.415,-43.282,178.738,5.943,149.437
C03070=1151.052,-107.165,-43.291,178.741,5.944,149.437
C03071=1151.047,-106.915,-43.300,178.742,5.944,149.436
C03072=1151.042,-106.666,-43.309,178.744,5.944,149.436
C03073=1151.036,-106.415,-43.319,178.746,5.944,149.435
C03074=1151.031,-106.166,-43.328,178.749,5.945,149.435
C03075=1151.025,-105.916,-43.336,178.751,5.945,149.434
C03076=1151.020,-105.667,-43.346,178.752,5.945,149.434
C03077=1151.015,-105.417,-43.355,178.755,5.946,149.433
C03078=1151.009,-105.167,-43.364,178.757,5.946,149.432
C03079=1151.004,-104.917,-43.373,178.759,5.946,149.432
C03080=1150.999,-104.667,-43.382,178.761,5.947,149.431
C03081=1150.994,-104.418,-43.391,178.763,5.947,149.431
C03082=1150.988,-104.167,-43.400,178.765,5.948,149.430
C03083=1150.983,-103.918,-43.409,178.767,5.948,149.430
C03084=1150.978,-103.668,-43.419,178.769,5.948,149.429
C03085=1150.973,-103.419,-43.428,178.771,5.949,149.429
C03086=1150.967,-103.169,-43.436,178.773,5.949,149.428
C03087=1150.961,-102.897,-43.447,178.776,5.949,149.428
C03088=1150.955,-102.625,-43.457,178.778,5.950,149.427
C03089=1150.949,-102.353,-43.467,178.780,5.950,149.426
C03090=1150.944,-102.080,-43.476,178.782,5.950,149.426
C03091=1150.939,-101.831,-43.486,178.784,5.951,149.425
C03092=1150.933,-101.581,-43.495,178.786,5.951,149.425
C03093=1150.928,-101.331,-43.504,178.789,5.952,149.424
C03094=1150.922,-101.081,-43.513,178.791,5.952,149.424
C03095=1150.918,-100.832,-43.523,178.792,5.952,149.423
C03096=1150.912,-100.582,-43.532,178.795,5.953,149.423
C03097=1150.906,-100.332,-43.541,178.797,5.953,149.422
C03098=1150.901,-100.083,-43.550,178.799,5.953,149.422
C03099=1150.895,-99.833,-43.560,178.801,5.954,149.421
C03100=1150.890,-99.583,-43.569,178.803,5.954,149.421
C03101=1150.885,-99.333,-43.578,178.805,5.954,149.420
C03102=1150.879,-99.083,-43.587,178.807,5.954,149.419
C03103=1150.874,-98.834,-43.597,178.809,5.955,149.419
C03104=1150.869,-98.584,-43.606,178.811,5.956,149.418
C03105=1150.863,-98.334,-43.615,178.813,5.956,149.418
C03106=1150.858,-98.085,-43.625,178.816,5.956,149.417
C03107=1150.853,-97.835,-43.634,178.818,5.957,149.417
C03108=1150.847,-97.585,-43.643,178.819,5.957,149.416
C03109=1150.842,-97.335,-43.652,178.822,5.957,149.416
C03110=1150.836,-97.085,-43.662,178.824,5.957,149.415
C03111=1150.831,-96.835,-43.671,178.826,5.958,149.415
C03112=1150.826,-96.586,-43.680,178.828,5.959,149.414
C03113=1150.820,-96.336,-43.690,178.830,5.958,149.413
C03114=1150.815,-96.086,-43.699,178.832,5.959,149.413
C03115=1150.810,-95.837,-43.709,178.834,5.960,149.412
C03116=1150.804,-95.587,-43.718,178.836,5.960,149.412
C03117=1150.799,-95.337,-43.727,178.839,5.960,149.411
C03118=1150.794,-95.087,-43.737,178.841,5.961,149.411
C03119=1150.788,-94.838,-43.746,178.843,5.961,149.410
C03120=1150.783,-94.587,-43.756,178.845,5.962,149.410
C03121=1150.778,-94.338,-43.765,178.847,5.961,149.409
C03122=1150.773,-94.088,-43.775,178.849,5.962,149.409
C03123=1150.768,-93.838,-43.785,178.851,5.963,149.408
C03124=1150.762,-93.588,-43.794,178.853,5.963,149.407
C03125=1150.756,-93.338,-43.803,178.855,5.963,149.407
C03126=1150.752,-93.089,-43.813,178.858,5.964,149.406
C03127=1150.746,-92.839,-43.822,178.859,5.964,149.406
C03128=1150.741,-92.589,-43.832,178.862,5.964,149.405
C03129=1150.735,-92.339,-43.842,178.864,5.965,149.405
C03130=1150.730,-92.090,-43.851,178.866,5.965,149.404
C03131=1150.724,-91.840,-43.861,178.868,5.966,149.404
C03132=1150.719,-91.591,-43.870,178.871,5.966,149.403
C03133=1150.714,-91.341,-43.879,178.872,5.966,149.403
C03134=1150.709,-91.091,-43.889,178.874,5.967,149.402
C03135=1150.703,-90.841,-43.898,178.877,5.967,149.401
C03136=1150.698,-90.591,-43.909,178.879,5.967,149.401
C03137=1150.693,-90.341,-43.918,178.881,5.968,149.400
C03138=1150.688,-90.092,-43.928,178.882,5.968,149.400
C03139=1150.682,-89.842,-43.937,178.885,5.968,149.399
C03140=1150.677,-89.592,-43.947,178.887,5.969,149.399
C03141=1150.671,-89.342,-43.957,178.889,5.969,149.398
C03142=1150.666,-89.093,-43.966,178.892,5.970,149.398
C03143=1150.660,-88.843,-43.976,178.894,5.970,149.397
C03144=1150.655,-88.594,-43.985,178.895,5.970,149.397
C03145=1150.649,-88.343,-43.995,178.898,5.971,149.396
C03146=1150.645,-88.094,-44.005,178.900,5.971,149.395
C03147=1150.640,-87.844,-44.015,178.902,5.971,149.395
C03148=1150.634,-87.594,-44.024,178.904,5.972,149.394
C03149=1150.629,-87.345,-44.034,178.907,5.973,149.394
C03150=1150.624,-87.095,-44.043,178.908,5.973,149.393
C03151=1150.618,-86.845,-44.053,178.910,5.973,149.393
C03152=1150.612,-86.596,-44.063,178.913,5.974,149.392
C03153=1150.608,-86.345,-44.073,178.915,5.974,149.392
C03154=1150.602,-86.096,-44.083,178.917,5.974,149.391
C03155=1150.597,-85.846,-44.092,178.919,5.975,149.391
C03156=1150.591,-85.596,-44.102,178.922,5.976,149.390
C03157=1150.587,-85.347,-44.112,178.923,5.976,149.389
C03158=1150.581,-85.097,-44.121,178.926,5.976,149.389
C03159=1150.576,-84.846,-44.132,178.928,5.977,149.388
C03160=1150.571,-84.597,-44.141,178.930,5.977,149.388
C03161=1150.565,-84.347,-44.151,178.932,5.977,149.387
C03162=1150.560,-84.098,-44.160,178.934,5.978,149.387
C03163=1150.555,-83.848,-44.171,178.936,5.978,149.386
C03164=1150.550,-83.598,-44.181,178.938,5.979,149.386
C03165=1150.544,-83.348,-44.190,178.941,5.979,149.385
C03166=1150.539,-83.099,-44.200,178.943,5.979,149.384
C03167=1150.533,-82.849,-44.210,178.945,5.980,149.384
C03168=1150.528,-82.599,-44.219,178.947,5.980,149.383
C03169=1150.523,-82.349,-44.230,178.950,5.981,149.383
C03170=1150.517,-82.100,-44.240,178.951,5.981,149.382
C03171=1150.513,-81.850,-44.250,178.954,5.982,149.382
C03172=1150.507,-81.600,-44.259,178.956,5.982,149.381
C03173=1150.501,-81.351,-44.269,178.958,5.982,149.381
C03174=1150.497,-81.101,-44.279,178.960,5.983,149.380
C03175=1150.491,-80.851,-44.290,178.962,5.983,149.380
C03176=1150.485,-80.601,-44.299,178.964,5.983,149.379
C03177=1150.480,-80.352,-44.309,178.967,5.984,149.378
C03178=1150.475,-80.102,-44.319,178.969,5.985,149.378
C03179=1150.470,-79.852,-44.329,178.971,5.985,149.377
C03180=1150.464,-79.602,-44.340,178.973,5.985,149.377
C03181=1150.459,-79.353,-44.349,178.975,5.986,149.376
C03182=1150.453,-79.103,-44.359,178.978,5.986,149.375
C03183=1150.448,-78.853,-44.369,178.979,5.986,149.375
C03184=1150.444,-78.604,-44.379,178.982,5.987,149.375
C03185=1150.438,-78.354,-44.389,178.984,5.987,149.374
C03186=1150.432,-78.104,-44.399,178.986,5.988,149.373
C03187=1150.427,-77.854,-44.409,178.988,5.988,149.373
C03188=1150.421,-77.604,-44.419,178.991,5.988,149.372
C03189=1150.417,-77.355,-44.429,178.993,5.989,149.372
C03190=1150.411,-77.105,-44.439,178.995,5.989,149.371
C03191=1150.405,-76.834,-44.451,178.997,5.989,149.370
C03192=1150.400,-76.562,-44.462,178.999,5.990,149.370
C03193=1150.394,-76.290,-44.472,179.002,5.991,149.369
C03194=1150.388,-76.020,-44.483,179.004,5.991,149.369
C03195=1150.383,-75.769,-44.494,179.007,5.992,149.368
C03196=1150.377,-75.520,-44.504,179.009,5.992,149.368
C03197=1150.372,-75.270,-44.514,179.011,5.992,149.367
C03198=1150.367,-75.021,-44.524,179.013,5.993,149.366
C03199=1150.362,-74.771,-44.534,179.016,5.994,149.366
C03200=1150.356,-74.521,-44.545,179.018,5.993,149.365
C03201=1150.351,-74.272,-44.555,179.020,5.994,149.365
C03202=1150.346,-74.021,-44.565,179.022,5.995,149.364
C03203=1150.341,-73.772,-44.575,179.025,5.995,149.364
C03204=1150.335,-73.523,-44.585,179.026,5.995,149.363
C03205=1150.330,-73.272,-44.596,179.029,5.996,149.363
C03206=1150.325,-73.023,-44.606,179.031,5.996,149.362
C03207=1150.319,-72.773,-44.616,179.033,5.996,149.361
C03208=1150.314,-72.523,-44.627,179.035,5.997,149.361
C03209=1150.308,-72.273,-44.637,179.038,5.997,149.360
C03210=1150.304,-72.024,-44.647,179.040,5.998,149.360
C03211=1150.299,-71.774,-44.657,179.041,5.998,149.359
C03212=1150.293,-71.524,-44.667,179.044,5.999,149.359
C03213=1150.287,-71.275,-44.678,179.046,5.999,149.358
C03214=1150.282,-71.025,-44.688,179.048,6.000,149.358
C03215=1150.277,-70.775,-44.698,179.051,6.000,149.357
C03216=1150.271,-70.526,-44.709,179.053,6.001,149.356
C03217=1150.266,-70.275,-44.719,179.055,6.001,149.356
C03218=1150.261,-70.026,-44.729,179.058,6.002,149.355
C03219=1150.255,-69.776,-44.740,179.059,6.002,149.355
C03220=1150.251,-69.526,-44.750,179.061,6.002,149.354
C03221=1150.245,-69.277,-44.760,179.064,6.003,149.354
C03222=1150.240,-69.027,-44.770,179.066,6.004,149.353
C03223=1150.235,-68.778,-44.781,179.069,6.004,149.352
C03224=1150.229,-68.528,-44.791,179.070,6.004,149.352
C03225=1150.224,-68.278,-44.802,179.073,6.005,149.351
C03226=1150.219,-68.028,-44.812,179.075,6.005,149.351
C03227=1150.214,-67.778,-44.823,179.078,6.006,149.350
C03228=1150.208,-67.528,-44.833,179.079,6.006,149.350
C03229=1150.202,-67.279,-44.843,179.082,6.006,149.349
C03230=1150.197,-67.029,-44.854,179.084,6.007,149.349
C03231=1150.192,-66.780,-44.865,179.086,6.008,149.348
C03232=1150.187,-66.530,-44.875,179.088,6.007,149.347
C03233=1150.182,-66.280,-44.885,179.090,6.008,149.347
C03234=1150.176,-66.030,-44.896,179.093,6.009,149.346
C03235=1150.171,-65.780,-44.906,179.095,6.009,149.346
C03236=1150.166,-65.531,-44.917,179.098,6.010,149.345
C03237=1150.161,-65.281,-44.928,179.100,6.010,149.344
C03238=1150.155,-65.031,-44.938,179.102,6.010,149.344
C03239=1150.150,-64.781,-44.949,179.104,6.011,149.344
C03240=1150.144,-64.532,-44.959,179.107,6.012,149.343
C03241=1150.140,-64.282,-44.970,179.109,6.012,149.342
C03242=1150.134,-64.033,-44.980,179.110,6.012,149.342
C03243=1150.129,-63.783,-44.990,179.113,6.013,149.341
C03244=1150.124,-63.533,-45.002,179.115,6.014,149.341
C03245=1150.118,-63.284,-45.012,179.118,6.014,149.340
C03246=1150.113,-63.034,-45.023,179.120,6.014,149.339
C03247=1150.108,-62.784,-45.033,179.122,6.015,149.339
C03248=1150.103,-62.534,-45.044,179.124,6.015,149.338
C03249=1150.097,-62.285,-45.054,179.127,6.016,149.338
C03250=1150.092,-62.035,-45.065,179.129,6.017,149.337
C03251=1150.086,-61.785,-45.076,179.131,6.016,149.337
C03252=1150.081,-61.535,-45.087,179.133,6.017,149.336
C03253=1150.076,-61.286,-45.097,179.136,6.017,149.335
C03254=1150.071,-61.036,-45.108,179.138,6.018,149.335
C03255=1150.065,-60.786,-45.119,179.140,6.019,149.334
C03256=1150.060,-60.536,-45.129,179.142,6.019,149.334
C03257=1150.055,-60.287,-45.140,179.144,6.019,149.333
C03258=1150.050,-60.037,-45.151,179.147,6.020,149.333
C03259=1150.045,-59.787,-45.161,179.149,6.021,149.332
C03260=1150.040,-59.538,-45.172,179.151,6.021,149.332
C03261=1150.034,-59.288,-45.183,179.154,6.022,149.331
C03262=1150.029,-59.038,-45.194,179.156,6.022,149.330
C03263=1150.023,-58.789,-45.204,179.158,6.023,149.330
C03264=1150.018,-58.539,-45.215,179.161,6.023,149.329
C03265=1150.014,-58.289,-45.226,179.163,6.024,149.329
C03266=1150.008,-58.039,-45.237,179.165,6.024,149.328
C03267=1150.003,-57.790,-45.248,179.167,6.024,149.328
C03268=1149.997,-57.540,-45.259,179.169,6.025,149.327
C03269=1149.992,-57.290,-45.270,179.172,6.025,149.326
C03270=1149.987,-57.041,-45.280,179.174,6.026,149.326
C03271=1149.982,-56.791,-45.291,179.177,6.026,149.325
C03272=1149.977,-56.541,-45.302,179.179,6.027,149.325
C03273=1149.971,-56.291,-45.312,179.180,6.027,149.324
C03274=1149.966,-56.041,-45.324,179.183,6.028,149.324
C03275=1149.960,-55.792,-45.334,179.185,6.028,149.323
C03276=1149.956,-55.542,-45.346,179.188,6.029,149.322
C03277=1149.950,-55.293,-45.356,179.190,6.030,149.322
C03278=1149.945,-55.043,-45.368,179.192,6.030,149.321
C03279=1149.940,-54.792,-45.378,179.194,6.030,149.321
C03280=1149.934,-54.544,-45.389,179.197,6.031,149.320
C03281=1149.929,-54.293,-45.400,179.199,6.031,149.320
C03282=1149.924,-54.044,-45.411,179.201,6.032,149.319
C03283=1149.919,-53.794,-45.423,179.204,6.033,149.319
C03284=1149.914,-53.544,-45.433,179.206,6.033,149.318
C03285=1149.908,-53.295,-45.444,179.208,6.033,149.317
C03286=1149.903,-53.045,-45.455,179.211,6.033,149.317
C03287=1149.897,-52.796,-45.466,179.213,6.034,149.316
C03288=1149.892,-52.546,-45.477,179.215,6.035,149.316
C03289=1149.888,-52.296,-45.488,179.218,6.035,149.315
C03290=1149.882,-52.047,-45.500,179.220,6.036,149.315
C03291=1149.877,-51.796,-45.510,179.222,6.036,149.314
C03292=1149.872,-51.547,-45.521,179.224,6.037,149.313
C03293=1149.867,-51.298,-45.532,179.226,6.037,149.313
C03294=1149.861,-51.047,-45.544,179.229,6.038,149.312
C03295=1149.855,-50.776,-45.556,179.231,6.039,149.312
C03296=1149.850,-50.506,-45.567,179.234,6.039,149.311
C03297=1149.844,-50.235,-45.579,179.236,6.039,149.310
C03298=1149.838,-49.965,-45.591,179.239,6.040,149.310
C03299=1149.833,-49.716,-45.602,179.241,6.040,149.309
C03300=1149.828,-49.466,-45.614,179.243,6.041,149.309
C03301=1149.822,-49.216,-45.625,179.246,6.042,149.308
C03302=1149.818,-48.966,-45.636,179.248,6.042,149.307
C03303=1149.812,-48.717,-45.648,179.250,6.042,149.307
C03304=1149.807,-48.467,-45.658,179.253,6.043,149.306
C03305=1149.801,-48.217,-45.670,179.255,6.044,149.306
C03306=1149.796,-47.967,-45.681,179.257,6.044,149.305
C03307=1149.791,-47.718,-45.692,179.260,6.045,149.305
C03308=1149.785,-47.468,-45.703,179.262,6.046,149.304
C03309=1149.781,-47.218,-45.715,179.265,6.046,149.303
C03310=1149.775,-46.968,-45.726,179.267,6.047,149.303
C03311=1149.770,-46.719,-45.737,179.268,6.047,149.303
C03312=1149.765,-46.469,-45.748,179.271,6.047,149.302
C03313=1149.760,-46.219,-45.760,179.273,6.048,149.301
C03314=1149.754,-45.970,-45.771,179.276,6.048,149.301
C03315=1149.749,-45.720,-45.783,179.278,6.049,149.300
C03316=1149.744,-45.471,-45.794,179.281,6.050,149.299
C03317=1149.739,-45.221,-45.804,179.283,6.050,149.299
C03318=1149.733,-44.971,-45.816,179.285,6.051,149.298
C03319=1149.728,-44.722,-45.827,179.288,6.052,149.298
C03320=1149.723,-44.472,-45.839,179.289,6.052,149.297
C03321=1149.718,-44.222,-45.850,179.292,6.052,149.297
C03322=1149.712,-43.973,-45.862,179.294,6.053,149.296
C03323=1149.707,-43.723,-45.873,179.297,6.053,149.295
C03324=1149.702,-43.473,-45.884,179.299,6.054,149.295
C03325=1149.697,-43.223,-45.896,179.301,6.055,149.294
C03326=1149.691,-42.974,-45.907,179.304,6.055,149.294
C03327=1149.686,-42.724,-45.919,179.306,6.056,149.293
C03328=1149.681,-42.474,-45.930,179.309,6.056,149.293
C03329=1149.676,-42.225,-45.942,179.311,6.057,149.292
C03330=1149.670,-41.975,-45.953,179.312,6.057,149.292
C03331=1149.666,-41.726,-45.965,179.315,6.058,149.291
C03332=1149.660,-41.475,-45.976,179.317,6.058,149.290
C03333=1149.655,-41.226,-45.987,179.320,6.059,149.290
C03334=1149.650,-40.976,-45.999,179.322,6.059,149.289
C03335=1149.644,-40.727,-46.010,179.325,6.060,149.289
C03336=1149.639,-40.477,-46.022,179.327,6.061,149.288
C03337=1149.634,-40.227,-46.033,179.329,6.061,149.288
C03338=1149.629,-39.977,-46.045,179.332,6.062,149.287
C03339=1149.624,-39.728,-46.056,179.334,6.063,149.286
C03340=1149.618,-39.478,-46.068,179.337,6.063,149.286
C03341=1149.613,-39.228,-46.080,179.339,6.064,149.285
C03342=1149.608,-38.979,-46.091,179.341,6.063,149.285
C03343=1149.603,-38.729,-46.103,179.343,6.064,149.284
C03344=1149.598,-38.479,-46.114,179.345,6.065,149.284
C03345=1149.592,-38.230,-46.126,179.348,6.065,149.283
C03346=1149.586,-37.980,-46.137,179.350,6.066,149.282
C03347=1149.582,-37.730,-46.149,179.353,6.067,149.282
C03348=1149.576,-37.481,-46.161,179.355,6.067,149.281
C03349=1149.572,-37.231,-46.172,179.358,6.068,149.281
C03350=1149.566,-36.981,-46.184,179.360,6.069,149.280
C03351=1149.560,-36.732,-46.195,179.362,6.069,149.280
C03352=1149.556,-36.483,-46.207,179.365,6.070,149.279
C03353=1149.550,-36.233,-46.219,179.367,6.071,149.278
C03354=1149.545,-35.983,-46.231,179.370,6.071,149.278
C03355=1149.540,-35.733,-46.242,179.372,6.072,149.277
C03356=1149.535,-35.483,-46.254,179.374,6.072,149.277
C03357=1149.529,-35.233,-46.266,179.376,6.072,149.276
C03358=1149.525,-34.984,-46.277,179.378,6.073,149.276
C03359=1149.519,-34.734,-46.289,179.381,6.073,149.275
C03360=1149.513,-34.485,-46.301,179.383,6.074,149.274
C03361=1149.509,-34.236,-46.313,179.386,6.075,149.274
C03362=1149.503,-33.986,-46.325,179.388,6.075,149.273
C03363=1149.498,-33.736,-46.337,179.391,6.076,149.273
C03364=1149.493,-33.486,-46.348,179.393,6.077,149.272
C03365=1149.488,-33.236,-46.360,179.395,6.077,149.271
C03366=1149.482,-32.986,-46.372,179.398,6.078,149.271
C03367=1149.478,-32.737,-46.384,179.400,6.079,149.270
C03368=1149.473,-32.487,-46.396,179.402,6.079,149.270
C03369=1149.467,-32.238,-46.407,179.405,6.080,149.269
C03370=1149.461,-31.988,-46.419,179.407,6.080,149.269
C03371=1149.457,-31.739,-46.431,179.409,6.081,149.268
C03372=1149.451,-31.489,-46.443,179.412,6.081,149.267
C03373=1149.446,-31.239,-46.455,179.414,6.082,149.267
C03374=1149.440,-30.989,-46.467,179.417,6.083,149.266
C03375=1149.436,-30.740,-46.479,179.419,6.083,149.266
C03376=1149.431,-30.490,-46.490,179.421,6.084,149.265
C03377=1149.425,-30.240,-46.502,179.424,6.085,149.265
C03378=1149.420,-29.990,-46.514,179.426,6.085,149.264
C03379=1149.415,-29.741,-46.526,179.429,6.086,149.263
C03380=1149.410,-29.491,-46.538,179.431,6.087,149.263
C03381=1149.405,-29.242,-46.550,179.434,6.087,149.262
C03382=1149.399,-28.992,-46.563,179.436,6.088,149.262
C03383=1149.394,-28.742,-46.575,179.437,6.088,149.261
C03384=1149.389,-28.493,-46.586,179.440,6.088,149.261
C03385=1149.384,-28.243,-46.598,179.442,6.089,149.260
C03386=1149.379,-27.993,-46.610,179.445,6.090,149.259
C03387=1149.373,-27.743,-46.622,179.447,6.090,149.259
C03388=1149.368,-27.494,-46.635,179.450,6.091,149.258
C03389=1149.363,-27.244,-46.647,179.452,6.092,149.258
C03390=1149.358,-26.995,-46.658,179.455,6.092,149.257
C03391=1149.353,-26.745,-46.671,179.457,6.093,149.257
C03392=1149.348,-26.495,-46.682,179.459,6.094,149.256
C03393=1149.342,-26.246,-46.695,179.462,6.094,149.255
C03394=1149.337,-25.996,-46.707,179.464,6.095,149.255
C03395=1149.332,-25.746,-46.719,179.467,6.095,149.254
C03396=1149.326,-25.497,-46.731,179.469,6.096,149.254
C03397=1149.322,-25.247,-46.743,179.471,6.096,149.253
C03398=1149.317,-24.998,-46.755,179.474,6.097,149.253
C03399=1149.311,-24.728,-46.768,179.477,6.098,149.252
C03400=1149.305,-24.458,-46.781,179.479,6.099,149.252
C03401=1149.300,-24.188,-46.795,179.482,6.100,149.251
C03402=1149.294,-23.918,-46.808,179.484,6.100,149.250
C03403=1149.289,-23.668,-46.820,179.487,6.101,149.250
C03404=1149.284,-23.418,-46.833,179.489,6.101,149.249
C03405=1149.278,-23.168,-46.844,179.491,6.102,149.248
C03406=1149.273,-22.919,-46.857,179.494,6.103,149.248
C03407=1149.268,-22.669,-46.869,179.496,6.103,149.247
C03408=1149.263,-22.420,-46.882,179.498,6.104,149.247
C03409=1149.257,-22.170,-46.893,179.501,6.104,149.246
C03410=1149.252,-21.920,-46.906,179.503,6.105,149.246
C03411=1149.247,-21.671,-46.919,179.506,6.106,149.245
C03412=1149.242,-21.421,-46.931,179.508,6.107,149.245
C03413=1149.236,-21.172,-46.943,179.511,6.107,149.244
C03414=1149.231,-20.922,-46.955,179.513,6.108,149.243
C03415=1149.226,-20.673,-46.968,179.515,6.109,149.243
C03416=1149.221,-20.422,-46.980,179.518,6.109,149.242
C03417=1149.216,-20.173,-46.992,179.520,6.110,149.242
C03418=1149.211,-19.923,-47.005,179.523,6.110,149.241
C03419=1149.205,-19.673,-47.017,179.525,6.111,149.241
C03420=1149.200,-19.424,-47.030,179.527,6.111,149.240
C03421=1149.195,-19.174,-47.041,179.530,6.113,149.239
C03422=1149.190,-18.925,-47.054,179.533,6.113,149.239
C03423=1149.185,-18.676,-47.067,179.535,6.114,149.238
C03424=1149.179,-18.426,-47.079,179.538,6.115,149.238
C03425=1149.175,-18.176,-47.092,179.540,6.115,149.237
C03426=1149.169,-17.926,-47.104,179.542,6.116,149.237
C03427=1149.164,-17.676,-47.116,179.545,6.117,149.236
C03428=1149.159,-17.427,-47.129,179.547,6.117,149.235
C03429=1149.154,-17.178,-47.141,179.550,6.118,149.235
C03430=1149.149,-16.928,-47.154,179.552,6.119,149.234
C03431=1149.143,-16.678,-47.166,179.554,6.119,149.234
C03432=1149.139,-16.428,-47.179,179.557,6.120,149.233
C03433=1149.133,-16.179,-47.192,179.559,6.120,149.232
C03434=1149.127,-15.929,-47.204,179.561,6.121,149.232
C03435=1149.122,-15.680,-47.216,179.564,6.122,149.231
C03436=1149.117,-15.430,-47.229,179.566,6.122,149.231
C03437=1149.113,-15.180,-47.242,179.568,6.123,149.230
C03438=1149.107,-14.930,-47.254,179.571,6.124,149.230
C03439=1149.102,-14.681,-47.266,179.573,6.124,149.229
C03440=1149.097,-14.432,-47.279,179.577,6.126,149.228
C03441=1149.092,-14.182,-47.292,179.579,6.126,149.228
C03442=1149.087,-13.932,-47.305,179.581,6.127,149.227
C03443=1149.081,-13.682,-47.317,179.584,6.128,149.227
C03444=1149.076,-13.433,-47.330,179.586,6.128,149.226
C03445=1149.071,-13.183,-47.342,179.588,6.129,149.226
C03446=1149.066,-12.934,-47.355,179.591,6.129,149.225
C03447=1149.061,-12.684,-47.368,179.593,6.130,149.224
C03448=1149.055,-12.434,-47.381,179.595,6.131,149.224
C03449=1149.050,-12.185,-47.394,179.598,6.131,149.223
C03450=1149.045,-11.935,-47.405,179.600,6.132,149.223
C03451=1149.040,-11.685,-47.418,179.603,6.133,149.222
C03452=1149.035,-11.436,-47.431,179.605,6.133,149.222
C03453=1149.029,-11.186,-47.444,179.608,6.135,149.221
C03454=1149.024,-10.937,-47.457,179.611,6.135,149.221
C03455=1149.020,-10.687,-47.470,179.613,6.136,149.220
C03456=1149.015,-10.438,-47.482,179.615,6.137,149.219
C03457=1149.009,-10.188,-47.495,179.618,6.137,149.219
C03458=1149.004,-9.939,-47.508,179.620,6.138,149.218
C03459=1148.999,-9.689,-47.521,179.622,6.139,149.218
C03460=1148.994,-9.439,-47.534,179.625,6.139,149.217
C03461=1148.989,-9.190,-47.546,179.627,6.140,149.217
C03462=1148.984,-8.940,-47.560,179.630,6.140,149.216
C03463=1148.978,-8.690,-47.572,179.632,6.141,149.215
C03464=1148.973,-8.440,-47.584,179.635,6.142,149.215
C03465=1148.968,-8.191,-47.597,179.637,6.143,149.214
C03466=1148.963,-7.941,-47.611,179.640,6.144,149.214
C03467=1148.958,-7.691,-47.623,179.642,6.144,149.213
C03468=1148.953,-7.443,-47.637,179.645,6.145,149.212
C03469=1148.947,-7.192,-47.650,179.647,6.146,149.212
C03470=1148.942,-6.943,-47.663,179.649,6.147,149.211
C03471=1148.937,-6.694,-47.675,179.652,6.147,149.211
C03472=1148.932,-6.443,-47.689,179.654,6.148,149.210
C03473=1148.927,-6.194,-47.701,179.657,6.149,149.210
C03474=1148.922,-5.945,-47.714,179.660,6.150,149.209
C03475=1148.916,-5.694,-47.728,179.662,6.150,149.208
C03476=1148.911,-5.445,-47.740,179.664,6.151,149.208
C03477=1148.906,-5.196,-47.753,179.667,6.151,149.207
C03478=1148.901,-4.945,-47.766,179.669,6.152,149.207
C03479=1148.896,-4.696,-47.779,179.672,6.153,149.206
C03480=1148.891,-4.447,-47.792,179.674,6.154,149.206
C03481=1148.886,-4.197,-47.806,179.677,6.155,149.205
C03482=1148.881,-3.948,-47.818,179.680,6.156,149.205
C03483=1148.875,-3.698,-47.832,179.682,6.156,149.204
C03484=1148.870,-3.448,-47.845,179.684,6.157,149.203
C03485=1148.865,-3.199,-47.857,179.687,6.158,149.203
C03486=1148.860,-2.949,-47.871,179.689,6.158,149.202
C03487=1148.855,-2.700,-47.884,179.691,6.159,149.202
C03488=1148.849,-2.450,-47.897,179.694,6.159,149.201
C03489=1148.845,-2.200,-47.910,179.697,6.161,149.201
C03490=1148.839,-1.951,-47.923,179.699,6.161,149.200
C03491=1148.834,-1.701,-47.936,179.702,6.162,149.199
C03492=1148.829,-1.452,-47.950,179.704,6.163,149.199
C03493=1148.824,-1.202,-47.963,179.706,6.163,149.198
C03494=1148.819,-0.952,-47.976,179.709,6.164,149.198
C03495=1148.813,-0.703,-47.989,179.711,6.165,149.197
C03496=1148.809,-0.453,-48.003,179.714,6.166,149.197
C03497=1148.803,-0.204,-48.016,179.717,6.167,149.196
C03498=1148.798,0.046,-48.029,179.719,6.168,149.196
C03499=1148.793,0.296,-48.042,179.722,6.168,149.195
C03500=1148.788,0.545,-48.055,179.724,6.169,149.194
C03501=1148.783,0.795,-48.069,179.726,6.169,149.194
C03502=1148.777,1.044,-48.082,179.729,6.171,149.193
C03503=1148.772,1.314,-48.097,179.732,6.171,149.193
C03504=1148.766,1.584,-48.111,179.734,6.172,149.192
C03505=1148.761,1.852,-48.125,179.737,6.173,149.191
C03506=1148.755,2.122,-48.139,179.740,6.174,149.191
C03507=1148.750,2.371,-48.152,179.742,6.175,149.190
C03508=1148.745,2.621,-48.166,179.745,6.175,149.190
C03509=1148.739,2.871,-48.179,179.747,6.176,149.189
C03510=1148.735,3.120,-48.193,179.750,6.177,149.189
C03511=1148.729,3.370,-48.206,179.752,6.178,149.188
C03512=1148.725,3.619,-48.220,179.754,6.179,149.187
C03513=1148.719,3.869,-48.233,179.757,6.179,149.187
C03514=1148.715,4.119,-48.246,179.759,6.180,149.186
C03515=1148.709,4.368,-48.260,179.763,6.181,149.186
C03516=1148.704,4.618,-48.273,179.765,6.182,149.185
C03517=1148.699,4.867,-48.287,179.767,6.182,149.184
C03518=1148.694,5.117,-48.300,179.770,6.183,149.184
C03519=1148.689,5.366,-48.314,179.772,6.184,149.183
C03520=1148.684,5.616,-48.327,179.774,6.184,149.183
C03521=1148.678,5.865,-48.341,179.777,6.186,149.182
C03522=1148.674,6.115,-48.354,179.780,6.187,149.182
C03523=1148.669,6.365,-48.368,179.782,6.187,149.181
C03524=1148.664,6.615,-48.381,179.785,6.188,149.181
C03525=1148.659,6.864,-48.395,179.787,6.189,149.180
C03526=1148.653,7.114,-48.408,179.790,6.190,149.179
C03527=1148.649,7.363,-48.422,179.792,6.191,149.179
C03528=1148.643,7.613,-48.435,179.795,6.191,149.178
C03529=1148.638,7.863,-48.450,179.797,6.192,149.178
C03530=1148.633,8.112,-48.462,179.800,6.192,149.177
C03531=1148.628,8.362,-48.476,179.803,6.194,149.177
C03532=1148.622,8.611,-48.490,179.805,6.195,149.176
C03533=1148.618,8.861,-48.503,179.807,6.195,149.176
C03534=1148.613,9.110,-48.518,179.809,6.196,149.175
C03535=1148.607,9.360,-48.531,179.812,6.197,149.174
C03536=1148.602,9.610,-48.545,179.815,6.198,149.174
C03537=1148.597,9.859,-48.558,179.818,6.199,149.173
C03538=1148.592,10.109,-48.572,179.820,6.199,149.173
C03539=1148.587,10.358,-48.586,179.822,6.200,149.172
C03540=1148.582,10.608,-48.599,179.825,6.201,149.172
C03541=1148.577,10.857,-48.613,179.827,6.202,149.171
C03542=1148.571,11.106,-48.627,179.830,6.203,149.170
C03543=1148.566,11.357,-48.641,179.832,6.204,149.170
C03544=1148.562,11.606,-48.654,179.835,6.204,149.169
C03545=1148.556,11.855,-48.668,179.838,6.206,149.169
C03546=1148.551,12.106,-48.682,179.840,6.206,149.168
C03547=1148.545,12.355,-48.696,179.842,6.207,149.168
C03548=1148.540,12.604,-48.710,179.845,6.207,149.167
C03549=1148.536,12.854,-48.723,179.848,6.209,149.167
C03550=1148.530,13.103,-48.737,179.850,6.209,149.166
C03551=1148.525,13.353,-48.751,179.853,6.210,149.165
C03552=1148.520,13.603,-48.765,179.855,6.211,149.165
C03553=1148.514,13.852,-48.779,179.858,6.212,149.164
C03554=1148.510,14.102,-48.792,179.860,6.213,149.164
C03555=1148.505,14.351,-48.807,179.863,6.214,149.163
C03556=1148.500,14.600,-48.820,179.865,6.214,149.163
C03557=1148.494,14.851,-48.834,179.868,6.216,149.162
C03558=1148.489,15.101,-48.848,179.870,6.216,149.162
C03559=1148.484,15.350,-48.862,179.873,6.217,149.161
C03560=1148.479,15.599,-48.876,179.875,6.218,149.160
C03561=1148.475,15.849,-48.890,179.878,6.219,149.160
C03562=1148.469,16.098,-48.904,179.881,6.220,149.159
C03563=1148.464,16.348,-48.918,179.883,6.221,149.159
C03564=1148.459,16.598,-48.932,179.886,6.221,149.158
C03565=1148.454,16.847,-48.946,179.888,6.223,149.158
C03566=1148.448,17.096,-48.960,179.891,6.223,149.157
C03567=1148.444,17.346,-48.974,179.893,6.224,149.157
C03568=1148.439,17.596,-48.989,179.896,6.224,149.156
C03569=1148.433,17.845,-49.003,179.899,6.226,149.155
C03570=1148.429,18.094,-49.016,179.901,6.227,149.155
C03571=1148.424,18.345,-49.030,179.903,6.227,149.154
C03572=1148.419,18.594,-49.044,179.906,6.229,149.154
C03573=1148.413,18.843,-49.058,179.909,6.229,149.153
C03574=1148.408,19.093,-49.072,179.911,6.230,149.153
C03575=1148.403,19.343,-49.087,179.914,6.231,149.152
C03576=1148.398,19.592,-49.101,179.916,6.232,149.152
C03577=1148.393,19.841,-49.115,179.919,6.233,149.151
C03578=1148.388,20.091,-49.129,179.921,6.234,149.150
C03579=1148.383,20.341,-49.143,179.923,6.234,149.150
C03580=1148.378,20.591,-49.158,179.927,6.236,149.149
C03581=1148.372,20.840,-49.171,179.929,6.236,149.149
C03582=1148.367,21.089,-49.186,179.931,6.237,149.148
C03583=1148.362,21.339,-49.200,179.934,6.239,149.148
C03584=1148.357,21.589,-49.214,179.937,6.239,149.147
C03585=1148.352,21.838,-49.228,179.939,6.240,149.147
C03586=1148.347,22.087,-49.242,179.941,6.241,149.146
C03587=1148.342,22.337,-49.257,179.944,6.242,149.145
C03588=1148.337,22.587,-49.271,179.947,6.243,149.145
C03589=1148.332,22.837,-49.285,179.949,6.243,149.144
C03590=1148.327,23.085,-49.300,179.952,6.245,149.144
C03591=1148.322,23.335,-49.314,179.955,6.245,149.143
C03592=1148.317,23.584,-49.328,179.957,6.246,149.143
C03593=1148.312,23.834,-49.343,179.960,6.247,149.142
C03594=1148.307,24.084,-49.357,179.962,6.248,149.142
C03595=1148.301,24.334,-49.372,179.964,6.249,149.141
C03596=1148.296,24.583,-49.386,179.968,6.250,149.140
C03597=1148.291,24.833,-49.400,179.970,6.251,149.140
C03598=1148.286,25.082,-49.415,179.972,6.252,149.139
C03599=1148.281,25.331,-49.429,179.975,6.252,149.139
C03600=1148.276,25.581,-49.444,179.978,6.254,149.138
C03601=1148.271,25.831,-49.458,179.980,6.254,149.138
C03602=1148.266,26.080,-49.472,179.982,6.255,149.137
C03603=1148.261,26.329,-49.486,179.985,6.257,149.137
C03604=1148.255,26.579,-49.502,179.988,6.257,149.136
C03605=1148.250,26.829,-49.516,179.990,6.258,149.135
C03606=1148.245,27.078,-49.530,179.993,6.259,149.135
C03607=1148.240,27.347,-49.546,179.996,6.260,149.134
C03608=1148.235,27.616,-49.562,179.998,6.262,149.134
C03609=1148.229,27.886,-49.577,-179.999,6.262,149.133
C03610=1148.224,28.154,-49.593,-179.996,6.263,149.132
C03611=1148.218,28.403,-49.607,-179.994,6.264,149.132
C03612=1148.214,28.652,-49.622,-179.991,6.265,149.132
C03613=1148.209,28.902,-49.636,-179.988,6.266,149.131
C03614=1148.203,29.152,-49.651,-179.986,6.267,149.130
C03615=1148.198,29.401,-49.666,-179.983,6.268,149.130
C03616=1148.193,29.651,-49.680,-179.981,6.269,149.129
C03617=1148.188,29.901,-49.695,-179.978,6.270,149.129
C03618=1148.183,30.150,-49.710,-179.975,6.271,149.128
C03619=1148.178,30.400,-49.724,-179.973,6.272,149.128
C03620=1148.173,30.650,-49.739,-179.970,6.272,149.127
C03621=1148.168,30.899,-49.754,-179.968,6.274,149.127
C03622=1148.163,31.149,-49.769,-179.965,6.275,149.126
C03623=1148.158,31.398,-49.783,-179.963,6.275,149.125
C03624=1148.153,31.647,-49.798,-179.960,6.277,149.125
C03625=1148.148,31.897,-49.812,-179.957,6.278,149.124
C03626=1148.142,32.146,-49.827,-179.955,6.278,149.124
C03627=1148.137,32.396,-49.842,-179.952,6.280,149.123
C03628=1148.133,32.645,-49.857,-179.950,6.280,149.123
C03629=1148.128,32.894,-49.871,-179.947,6.282,149.122
C03630=1148.122,33.144,-49.886,-179.944,6.283,149.122
C03631=1148.117,33.393,-49.901,-179.942,6.283,149.121
C03632=1148.112,33.643,-49.915,-179.939,6.285,149.120
C03633=1148.107,33.893,-49.931,-179.937,6.285,149.120
C03634=1148.102,34.142,-49.945,-179.934,6.286,149.119
C03635=1148.097,34.391,-49.960,-179.931,6.288,149.119
C03636=1148.092,34.641,-49.975,-179.929,6.288,149.118
C03637=1148.087,34.891,-49.990,-179.926,6.290,149.118
C03638=1148.082,35.140,-50.004,-179.924,6.290,149.117
C03639=1148.077,35.390,-50.020,-179.921,6.291,149.117
C03640=1148.072,35.639,-50.034,-179.918,6.293,149.116
C03641=1148.066,35.889,-50.049,-179.916,6.293,149.116
C03642=1148.062,36.138,-50.064,-179.914,6.294,149.115
C03643=1148.057,36.388,-50.079,-179.910,6.295,149.114
C03644=1148.052,36.638,-50.095,-179.908,6.296,149.114
C03645=1148.047,36.887,-50.109,-179.905,6.298,149.113
C03646=1148.042,37.137,-50.125,-179.903,6.298,149.113
C03647=1148.037,37.386,-50.140,-179.901,6.299,149.112
C03648=1148.032,37.636,-50.154,-179.897,6.300,149.112
C03649=1148.027,37.885,-50.169,-179.895,6.301,149.111
C03650=1148.022,38.135,-50.184,-179.892,6.303,149.111
C03651=1148.016,38.384,-50.199,-179.890,6.303,149.110
C03652=1148.012,38.633,-50.214,-179.888,6.304,149.110
C03653=1148.006,38.883,-50.229,-179.884,6.305,149.109
C03654=1148.001,39.132,-50.244,-179.882,6.306,149.109
C03655=1147.996,39.382,-50.260,-179.880,6.308,149.108
